	//iOptProportionalGainFor4
		aTransferPackages[15].iChannel := iParameterSet;
		aTransferPackages[15].iAddressedTarget := 8;
		aTransferPackages[15].iIndex := 249;
		
	// define end of parameter list to be uploaded by setting all variables to 0 (end criterion for FB_Upload_Multiple_Parameters)
		aTransferPackages[16].iChannel := 0;
		aTransferPackages[16].iAddressedTarget := 0;
		aTransferPackages[16].iIndex := 0;
//-----------------------------------------------------------------------------------------------------------

// Read the current status of the the motion terminal
	fbreadbitsfromword(wData:= awBusDataFromVTEM[0], iStartBit:=0, iEndBit:= 5, iValue=> iCurrentValveMode, xError=> );				// read current valve mode
//-----------------------------------------------------------------------------------------------------------

// Transition: Aborting condition when xAbort is TRUE in all States except "IDLE" , "ABORTING" and "RESETTING"
	IF xAbort = TRUE AND NOT(iState = 10 AND xExecute = FALSE) AND iState <> 80 AND iState <> 100 THEN
		xStateChange := TRUE;	// Leaving current state
		iState := 80;	// Choosing next state, here: ABORTING
	END_IF
//-----------------------------------------------------------------------------------------------------------

// local state machine
	CASE iState OF
		10:	// IDLE
			// code that is executed only in the first cycle of this state
				IF xStateChange = TRUE THEN
					xStateChange := FALSE;
					iResponse := eTransferResponse.ready_for_new_transfer;
					xDone := FALSE;
					xError := FALSE;
					xBusy := FALSE;
					xAborted := FALSE;
				END_IF
			//-----------------------------------------------------------------------------------------------------------
			
			// code that is repeated every cycle in this state
				iCommandNumber := 0;
			//-----------------------------------------------------------------------------------------------------------
			
			// Transition
			IF xExecute = TRUE THEN
				xStateChange := TRUE;
				iState := 20;
			END_IF
			//-----------------------------------------------------------------------------------------------------------
		
		20:	// RESETTING VALVE MODE TO 61
			// code that is executed only in the first cycle of this state
				IF xStateChange = TRUE THEN
					xStateChange := FALSE;
					iResponse := eTransferResponse.preparing_transfer;
					xDone := FALSE;
					xError := FALSE;
					xBusy := TRUE;
					xAborted := FALSE;
				END_IF
			//-----------------------------------------------------------------------------------------------------------
			
			// code that is repeated every cycle in this state	
				IF iCurrentValveMode = 63 THEN
					iCommandNumber := 5;	// exit transfer mode
				ELSIF iCurrentValveMode <> 61 AND iCurrentValveMode <> 63 THEN
					iCommandNumber := 6;	// stop running motion apps
				END_IF 
			//-----------------------------------------------------------------------------------------------------------
			
			// Transition
				IF iCurrentValveMode = 61 THEN
					xStateChange := TRUE;	// Leave this state
					iState := 30;
					iCommandNumber := 30;			
				END_IF
			//-----------------------------------------------------------------------------------------------------------
		
		30:	// READING PARAMETER VALUES
			// code that is executed only in the first cycle of this state
				IF xStateChange = TRUE THEN
					xStateChange := FALSE;
					iResponse := eTransferResponse.transferring;
					xDone := FALSE;
					xError := FALSE;
					xBusy := TRUE;
					xAborted := FALSE;
				END_IF
			//-----------------------------------------------------------------------------------------------------------
			
			// code that is repeated every cycle in this state
				iCommandNumber := 30;		// read parameter values
			//-----------------------------------------------------------------------------------------------------------
			
			// Transition
				IF fbuploadMultipleParameters.xExecute = TRUE AND fbuploadMultipleParameters.xUploadDone = TRUE AND fbuploadMultipleParameters.xUploadError = FALSE THEN	// Upload Done
					xStateChange := TRUE;
					iState := 40;	// Write parameter values to outputs
				ELSIF fbuploadMultipleParameters.xExecute = TRUE AND fbuploadMultipleParameters.xUploadDone = FALSE AND fbuploadMultipleParameters.xUploadError = TRUE THEN	// Error during update
					xStateChange := TRUE;
					iState := 70;	// ERROR
					iResponse := fbuploadMultipleParameters.iResponse;
				END_IF
			//-----------------------------------------------------------------------------------------------------------
		
		40:	// WRITE PARAMETER VALUES TO OUTPUTS
			// code that is executed only in the first cycle of this state
				IF xStateChange = TRUE THEN
					xStateChange := FALSE;
					iResponse := eTransferResponse.transferring;
					xDone := FALSE;
					xError := FALSE;
					xBusy := TRUE;
					xAborted := FALSE;
				END_IF
			//-----------------------------------------------------------------------------------------------------------
			
			// code that is repeated every cycle in this state
				iTubingLengthAt2			:= aTransferPackages[0].iTransferValue;
				iTubingLengthAt4			:= aTransferPackages[1].iTransferValue;
				iTubingInnerDiameterAt2		:= aTransferPackages[2].iTransferValue;
				iTubingInnerDiameterAt4		:= aTransferPackages[3].iTransferValue;
				iDriveType					:= aTransferPackages[4].iTransferValue;
				iDriveStroke				:= aTransferPackages[5].iTransferValue;
				iInstallationPositionDrive	:= aTransferPackages[6].iTransferValue;
				iLoadRetracting				:= aTransferPackages[7].iTransferValue;
				iLoadAdvancing				:= aTransferPackages[8].iTransferValue;
				iMomentOfInertiaRetracting	:= aTransferPackages[9].iTransferValue;
				iMomentOfInertiaAdvancing	:= aTransferPackages[10].iTransferValue;
				iSoftStartFunction			:= aTransferPackages[11].iTransferValue;
				iInPortRetracted_optional	:= aTransferPackages[12].iTransferValue;
				iInPortAdvanced_optional	:= aTransferPackages[13].iTransferValue;
				iOptProportionalGainFor2	:= aTransferPackages[14].iTransferValue;
				iOptProportionalGainFor4	:= aTransferPackages[15].iTransferValue;
			//-----------------------------------------------------------------------------------------------------------
			
			// Transition
				xStateChange := TRUE;
				iState := 50;
				iCommandNumber := 40;
			//-----------------------------------------------------------------------------------------------------------
		
		50:	// DONE
			// code that is executed only in the first cycle of this state
				IF xStateChange = TRUE THEN
					xStateChange := FALSE;
					iResponse := eTransferResponse.transfer_successful;
					xDone := TRUE;
					xError := FALSE;
					xBusy := FALSE;
					xAborted := FALSE;
				END_IF
			//-----------------------------------------------------------------------------------------------------------
			
			// code that is repeated every cycle in this state	
				IF fbuploadMultipleParameters.xExecute = FALSE  AND fbuploadMultipleParameters.xUploadDone = FALSE AND fbuploadMultipleParameters.xUploadError = FALSE AND iCurrentValveMode = 63 THEN		//FB_UploadMultipleParameters was reset
					iCommandNumber := 5;	// exit transfer mode
				END_IF
			//-----------------------------------------------------------------------------------------------------------
			
			// Transition
				IF fbuploadMultipleParameters.xExecute = FALSE  AND fbuploadMultipleParameters.xUploadDone = FALSE AND fbuploadMultipleParameters.xUploadError = FALSE AND xExecute = FALSE THEN
					xStateChange := TRUE;
					iState := 100;
				END_IF
			//-----------------------------------------------------------------------------------------------------------
			
		70:	// ERROR
			// code that is executed only in the first cycle of this state
				IF xStateChange = TRUE THEN
					xStateChange := FALSE;
					//iResponse := eTransferResponse.communication_failed;	// set within the transition of the last state
					xDone := FALSE;
					xError := TRUE;
					xBusy := FALSE;
					xAborted := FALSE;
				END_IF
			//-----------------------------------------------------------------------------------------------------------
			
			// code that is repeated every cycle in this state	
			//-----------------------------------------------------------------------------------------------------------
			
			// Transition
				IF xExecute = FALSE AND xAbort = FALSE THEN
					xStateChange := TRUE;
					iState := 100;
				END_IF
			//-----------------------------------------------------------------------------------------------------------
			
		80:	// ABORTING
			// code that is executed only in the first cycle of this state
				IF xStateChange = TRUE THEN
					xStateChange := FALSE;
					iResponse := eTransferResponse.aborting;
					xBusy := FALSE;
					xDone := FALSE;
					xError := FALSE;
					xAborted := TRUE;
				END_IF
			//-----------------------------------------------------------------------------------------------------------
			
			// code that is repeated every cycle in this state
				IF iCurrentValveMode = 63 THEN
					iCommandNumber := 5;	// exit transfer mode
				ELSIF iCurrentValveMode <> 61 AND iCurrentValveMode <> 63 THEN
					iCommandNumber := 6;	// stop running motion apps
				ELSE
					iCommandNumber := 0; 
				END_IF
			//-----------------------------------------------------------------------------------------------------------
			
			// Transition
				IF xAbort = FALSE AND xExecute = FALSE AND iCurrentValveMode = 61 THEN
					xStateChange := TRUE;
					iState := 100;
				END_IF
			//-----------------------------------------------------------------------------------------------------------

		100:	// RESETTING FUNCTION BLOCK AND VALVE
			// code that is executed only in the first cycle of this state
				IF xStateChange = TRUE THEN
					xStateChange := FALSE;
					iResponse := eTransferResponse.resetting;
					xDone := FALSE;
					xError := FALSE;
					xBusy := FALSE;
					xAborted := FALSE;
				END_IF
			//-----------------------------------------------------------------------------------------------------------
			
			// code that is repeated every cycle in this state	
				IF iCurrentValveMode = 63 THEN
					iCommandNumber := 5;	// exit transfer mode
				ELSIF iCurrentValveMode <> 61 AND iCurrentValveMode <> 63 THEN
					iCommandNumber := 6;	// stop running motion apps
				END_IF
				
				// reset funktion block fbreadmultipleparameters
				// not done via command number because this is used to reset valve
					fbuploadMultipleParameters(
						awBusDataFromVTEM:= awBusDataFromVTEM, 
						awBusDataToVTEM:= awBusDataToVTEM, 
						xExecute:= FALSE, 
						iResponse=> , 
						iCurrentValue=> , 
						xUploadDone=> , 
						xUploadError=> , 
						aTransferPackages:= aTransferPackages);
				
				// reset parameter outputs
					iParameterSet				:= 1;

					iTubingLengthAt2			:= 0;
					iTubingLengthAt4			:= 0;
					iTubingInnerDiameterAt2		:= 0;
					iTubingInnerDiameterAt4		:= 0;
					iDriveType					:= 0;
					iDriveStroke				:= 0;
					iInstallationPositionDrive	:= 0;
					iLoadRetracting				:= 0;
					iLoadAdvancing				:= 0;
					iMomentOfInertiaRetracting	:= 0;
					iMomentOfInertiaAdvancing	:= 0;
					iSoftStartFunction			:= 0;
					iInPortRetracted_optional	:= 0;
					iInPortAdvanced_optional	:= 0;
					iOptProportionalGainFor2	:= 0;
					iOptProportionalGainFor4	:= 0;
				
				// reset parameter array
					FOR iCounterResetArray := 0 TO 100 BY 1 DO
						aTransferPackages[iCounterResetArray].iChannel := 0;
						aTransferPackages[iCounterResetArray].iAddressedTarget := 0;
						aTransferPackages[iCounterResetArray].iIndex := 0;
						aTransferPackages[iCounterResetArray].iTransferValue := 0;
					END_FOR
					
					iCounterResetArray := 0;
					xFirstCycle := TRUE;
			//-----------------------------------------------------------------------------------------------------------
			
			// Transition
				IF iCurrentValveMode = 61 THEN
					iCommandNumber := 6; // Last command to send before the FB is in IDLE
					xStateChange := TRUE;
					iState := 10;
				END_IF
			//-----------------------------------------------------------------------------------------------------------
			
	END_CASE
//-----------------------------------------------------------------------------------------------------------

// Command section
	CASE iCommandNumber OF
		0:	// IDLE
			;
		
		5:	// EXIT TRANSFER MODE
			fbwritevaluetoword(iValue:=63, iStartBit:=0, iEndBit:=5, wDataWord:=awBusDataToVTEM[0], xError=> );							// Valve Mode = 63
			fbwritevaluetoword(iValue:=0, iStartBit:=6, iEndBit:=7, wDataWord:=awBusDataToVTEM[0], xError=> );							// 0 (unused)
			fbwritevaluetoword(iValue:=0, iStartBit:=8, iEndBit:=12, wDataWord:=awBusDataToVTEM[0], xError=> );							// Channel = 0 (ignored)
			fbwritevaluetoword(iValue:=3, iStartBit:=13, iEndBit:=15, wDataWord:=awBusDataToVTEM[0], xError=> );						// Transfer Control = 3 (Exit transfer mode)
			fbwritevaluetoword(iValue:=0, iStartBit:=0, iEndBit:=7, wDataWord:=awBusDataToVTEM[1], xError=> );							// Addressed Target = 0 (ignored)
			fbwritevaluetoword(iValue:=0, iStartBit:=8, iEndBit:=15, wDataWord:=awBusDataToVTEM[1], xError=> );							// Index = 0 (ignored)
			fbwritevaluetoword(iValue:=0, iStartBit:=0, iEndBit:=15, wDataWord:=awBusDataToVTEM[2], xError=> );							// Value = 0 (ignored)
			
		6:	// STOP RUNNING MOTION APP
			fbwritevaluetoword(iValue:=61, iStartBit:=0, iEndBit:=5, wDataWord:=awBusDataToVTEM[0], xError=> );							// Valve Mode = 61 (stop)
			fbwritevaluetoword(iValue:=0, iStartBit:=6, iEndBit:=7, wDataWord:=awBusDataToVTEM[0], xError=> );							// App Control = 0 (unused)
			fbwritevaluetoword(iValue:=0, iStartBit:=8, iEndBit:=15, wDataWord:=awBusDataToVTEM[0], xError=> );							// App Option = 0 (unused)
			fbwritevaluetoword(iValue:=0, iStartBit:=0, iEndBit:=15, wDataWord:=awBusDataToVTEM[1], xError=> );							// Setpoint Value 1 = 0 (unused)
			fbwritevaluetoword(iValue:=0, iStartBit:=0, iEndBit:=15, wDataWord:=awBusDataToVTEM[2], xError=> );							// Setpoint Value 2 = 0 (unused)
		
		30:	// RUN FB_UPLOADMULTIPLEPARAMETERS
			fbuploadMultipleParameters(
				awBusDataFromVTEM:= awBusDataFromVTEM, 
				awBusDataToVTEM:= awBusDataToVTEM, 
				xExecute:= TRUE, 
				iResponse=> , 
				iCurrentValue=> , 
				xUploadDone=> , 
				xUploadError=> , 
				aTransferPackages:= aTransferPackages);

		40:	// RESET FB_UPLOADMULTIPLEPARAMETERS
			fbuploadMultipleParameters(
				awBusDataFromVTEM:= awBusDataFromVTEM, 
				awBusDataToVTEM:= awBusDataToVTEM, 
				xExecute:= FALSE, 
				iResponse=> , 
				iCurrentValue=> , 
				xUploadDone=> , 
				xUploadError=> , 
				aTransferPackages:= aTransferPackages);
	END_CASE
//-----------------------------------------------------------------------------------------------------------

END_FUNCTION_BLOCK

// Transfermode/specific_MA_config/FB_Read_config_MA_10
/// This function block can be used to upload the configuration of Motion App 10 ("Flow control").
/// The specific parameters of this Motion App are the outputs of this FB
/// The function block uses the transfer mode to read this configuration from the Motion Terminal
/// and indicates the state of the upload process at the output iResponse.

FUNCTION_BLOCK FB_Read_config_MA_10
VAR_INPUT
	awBusDataFromVTEM 				: ARRAY [0..2] OF WORD;		// array of 3 words of process data received from the Motion Terminal
END_VAR
	
VAR_IN_OUT
	awBusDataToVTEM 				: ARRAY [0..2] OF WORD; 	// array of 3 words of process data sent to the Motion Terminal
END_VAR

VAR_INPUT
	xExecute 						: BOOL; 					// rising edge starts the reading process, falling edge resets the function block after reading is done
	xAbort							: BOOL;						// rising edge aborts the reading process
	iParameterSet					: INT := 1; 				// the parameter set to be read from, 1 by default
END_VAR                     		

VAR_OUTPUT                  		
	// system parameters
		iOperatingMedium			: eMA10OperatingMedium;		// Type and condition of the operating medium (values see eMA10OperatingMedium)
		iInPortFlowRate2_optional	: INT;						// Sensor port for flow rate at (2) (required for closed-loop controlled operating mode, value is number of the slot (beginning from 0 and including valve slots) * 10 + number of the port 
		iInPortFlowRate4_optional	: INT;						// Sensor port for flow rate at (4) (required for closed-loop controlled operating mode, value is number of the slot (beginning from 0 and including valve slots) * 10 + number of the port
		iInPortRetracted_optional	: INT;						// Sensor port for detection of end position at pressurisation of outlet port 2 (retracted), value is number of the slot (beginning from 0 and including valve slots) * 10 + number of the port
		iInPortAdvanced_optional	: INT;						// Sensor port for detection of end position at pressurisation of outlet port 4 (advanced), value is number of the slot (beginning from 0 and including valve slots) * 10 + number of the port

	// application parameters
		iCharacteristicAt2			: INT;						// Control characteristic, outlet port (2) (0 = "fast" (short tubes), 1 = medium (medium length tubes), 2 = "universal" (esp. long tubes), 3 = defined by tuning parameters (only if closed-loop control is activated for outlet port (2)))
		iCharacteristicAt4			: INT;						// Control characteristic, outlet port (4) (0 = "fast" (short tubes), 1 = medium (medium length tubes), 2 = "universal" (esp. long tubes), 3 = defined by tuning parameters (only if closed-loop control is activated for outlet port (4)))
		iOperatingMode				: INT;						// Operating mode of the Motion App (0 = (2) and (4) open-loop controlled; 1 = (2) open-loop, (4) closed-loop; 2 = (2) closed-loop, (4) open-loop; 3 = (2) and (4) closed-loop controlled) 
		xClosedLoopControl2			: BOOL;						// TRUE indicates closed-loop control for outlet port (2), FALSE is open-loop controlled operation (information is also part of parameter "iOperatingMode" and separated into an extra output for user comfort)
		xClosedLoopControl4			: BOOL;						// TRUE indicates closed-loop control for outlet port (4), FALSE is open-loop controlled operation (information is also part of parameter "iOperatingMode" and separated into an extra output for user comfort)
		
	// tuning parameters
		iOptProportionalGainFor2	: INT;						// Optional tuning parameter for the customized proportional element of the PID modulator at outlet port (2) [1 digit = 0.01 g/s/bar]
		iOptIntegralGainFor2		: INT;						// Optional tuning parameter for the customized integral element of the PID modulator at outlet port (2) [1 digit = 0.01 g/s²/bar]
		iOptRedFeedforwContrRate2	: INT;						// Optional tuning parameter for reduction of feedforward control rate of 100% for outlet port (2) [1 digit = 1%]
		iOptBoostSetpointReach2		: INT;						// Optional tuning parameter for boost to reach the setpoint value for outlet port (2) earlier, but with higher overshoot [1 digit = 1%] 
		iOptOffsetTargFRLimitInfo2	: INT;						// Optional tuning parameter for offset on the threshold value of 95% of the possible relative flow at outlet port (2) for feedback in app state, bit 5 [1 digit = 1%]
		iOptOffsetMinConsSetp2		: INT;						// Optional tuning parameter for offset to the threshold value of 25 l/min, below which a target flow rate for outlet port (2) is not considered [1 digit = 1 l/min]

		iOptProportionalGainFor4	: INT;						// Optional tuning parameter for the customized proportional element of the PID modulator at outlet port (4) [1 digit = 0.01 g/s/bar]
		iOptIntegralGainFor4		: INT;						// Optional tuning parameter for the customized integral element of the PID modulator at outlet port (4) [1 digit = 0.01 g/s²/bar]
		iOptRedFeedforwContrRate4	: INT;						// Optional tuning parameter for reduction of feedforward control rate of 100% for outlet port (4) [1 digit = 1%]
		iOptBoostSetpointReach4		: INT;						// Optional tuning parameter for boost to reach the setpoint value for outlet port (4) earlier, but with higher overshoot [1 digit = 1%] 
		iOptOffsetTargFRLimitInfo4	: INT;						// Optional tuning parameter for offset on the threshold value of 95% of the possible relative flow at outlet port (4) for feedback in app state, bit 5 [1 digit = 1%]
		iOptOffsetMinConsSetp4		: INT;						// Optional tuning parameter for offset to the threshold value of 25 l/min, below which a target flow rate for outlet port (4) is not considered [1 digit = 1 l/min]
		
	// function block response
		iResponse 					: eTransferResponse; 		// returns the status of the upload process
		xBusy						: BOOL;						// TRUE as long as the upload process is running
		xDone 						: BOOL; 					// indicates whether the upload was successfull
		xError 						: BOOL; 					// indicates whether an error occurred during the transfer
		xAborted					: BOOL;						// TRUE if the function block was canceled by xAbort	
END_VAR

VAR
	iState							: INT := 10;
	xStateChange					: BOOL;
	iCommandNumber					: INT;
	xFirstCycle						: BOOL := TRUE;				// indicator for the first cycle of the function block
	iParameterSetFC					: INT;						// value on input iParameterSet during first cycle
	
	aTransferPackages				: ARRAY [0..100] OF stTransferPackage;
	fbreadbitsfromword				: FB_Read_Bits_From_Word;
	fbuploadMultipleParameters 		: FB_Upload_Multiple_Parameters;
	fbWriteValueToWord 				: FB_Write_Value_To_Word;

	iCounterResetArray				: INT;

	iCurrentValveMode				: INT;						//
END_VAR

(*****************************************************************************************************

Festo SE & Co. KG, Esslingen
Copyright (c) 2021. All rights reserved.

Product:            Motion Terminal VTEM
Description:        Function Block to upload the parameters for Motion App 10 from the Motion Terminal

Object version:     2.00
Last change:        2021-07
======================================================================================================
                                       H I S T O R Y
======================================================================================================
Version:            2.00
Date:               2021-07
Change/Activity:    - created (#3872357)
Release:            3.5.7.237 (CODESYS 3.5.7.2, Lib version 3.7)
Author:             JEBU
======================================================================================================

*****************************************************************************************************)

// pre-check of the value for the parameter set
	IF xExecute = TRUE AND (iParameterSet < 1 OR iParameterSet > 5) THEN		// invalid input for the parameter set
		xDone := FALSE; 
		xError := TRUE; 
		iResponse := eTransferResponse.invalid_ParameterSet;
		xStateChange := TRUE;
		iState := 70;	// ERROR
	END_IF
//-----------------------------------------------------------------------------------------------------------

// check if iParameterSet was changed
	IF xExecute = TRUE AND xFirstCycle = TRUE THEN
		xFirstCycle := FALSE;
		iParameterSetFC := iParameterSet;
	END_IF
	
	IF xExecute = TRUE AND iParameterSet <> iParameterSetFC THEN
		xStateChange := TRUE;
		iState := 70;
		iResponse := eTransferResponse.FB_needs_rising_edge_xExecute;
	END_IF
//-----------------------------------------------------------------------------------------------------------

// WRITE PARAMETER INDICES INTO ARRAY
	//iOperatingMedium
		aTransferPackages[0].iChannel := iParameterSet;
		aTransferPackages[0].iAddressedTarget := 10;
		aTransferPackages[0].iIndex := 42;
	
	//iInPortFlowRate2_optional
		aTransferPackages[1].iChannel := iParameterSet;
		aTransferPackages[1].iAddressedTarget := 10;
		aTransferPackages[1].iIndex := 81;

	//iInPortFlowRate4_optional
		aTransferPackages[2].iChannel := iParameterSet;
		aTransferPackages[2].iAddressedTarget := 10;
		aTransferPackages[2].iIndex := 82;
	
	//iInPortRetracted_optional
		aTransferPackages[3].iChannel := iParameterSet;
		aTransferPackages[3].iAddressedTarget := 10;
		aTransferPackages[3].iIndex := 70;
	
	//iInPortAdvanced_optional
		aTransferPackages[4].iChannel := iParameterSet;
		aTransferPackages[4].iAddressedTarget := 10;
		aTransferPackages[4].iIndex := 71;
	
	//iCharacteristicAt2
		aTransferPackages[5].iChannel := iParameterSet;
		aTransferPackages[5].iAddressedTarget := 10;
		aTransferPackages[5].iIndex := 220;
	
	//iCharacteristicAt4
		aTransferPackages[6].iChannel := iParameterSet;
		aTransferPackages[6].iAddressedTarget := 10;
		aTransferPackages[6].iIndex := 221;
	
	//iOperatingMode
		aTransferPackages[7].iChannel := iParameterSet;
		aTransferPackages[7].iAddressedTarget := 10;
		aTransferPackages[7].iIndex := 223;
	
	//iOptProportionalGainFor2
		aTransferPackages[8].iChannel := iParameterSet;
		aTransferPackages[8].iAddressedTarget := 10;
		aTransferPackages[8].iIndex := 230;
	
	//iOptIntegralGainFor2
		aTransferPackages[9].iChannel := iParameterSet;
		aTransferPackages[9].iAddressedTarget := 10;
		aTransferPackages[9].iIndex := 231;
	
	//iOptRedFeedforwContrRate2
		aTransferPackages[10].iChannel := iParameterSet;
		aTransferPackages[10].iAddressedTarget := 10;
		aTransferPackages[10].iIndex := 232;
	
	//iOptBoostSetpointReach2
		aTransferPackages[11].iChannel := iParameterSet;
		aTransferPackages[11].iAddressedTarget := 10;
		aTransferPackages[11].iIndex := 233;
	
	//iOptOffsetTargFRLimitInfo2
		aTransferPackages[12].iChannel := iParameterSet;
		aTransferPackages[12].iAddressedTarget := 10;
		aTransferPackages[12].iIndex := 234;
	
	//iOptOffsetMinConsSetp2
		aTransferPackages[13].iChannel := iParameterSet;
		aTransferPackages[13].iAddressedTarget := 10;
		aTransferPackages[13].iIndex := 235;
	
	//iOptProportionalGainFor4
		aTransferPackages[14].iChannel := iParameterSet;
		aTransferPackages[14].iAddressedTarget := 10;
		aTransferPackages[14].iIndex := 240;
	
	//iOptIntegralGainFor4
		aTransferPackages[15].iChannel := iParameterSet;
		aTransferPackages[15].iAddressedTarget := 10;
		aTransferPackages[15].iIndex := 241;
	
	//iOptRedFeedforwContrRate4
		aTransferPackages[16].iChannel := iParameterSet;
		aTransferPackages[16].iAddressedTarget := 10;
		aTransferPackages[16].iIndex := 242;
	
	//iOptBoostSetpointReach4
		aTransferPackages[17].iChannel := iParameterSet;
		aTransferPackages[17].iAddressedTarget := 10;
		aTransferPackages[17].iIndex := 243;
	
	//iOptOffsetTargFRLimitInfo4
		aTransferPackages[18].iChannel := iParameterSet;
		aTransferPackages[18].iAddressedTarget := 10;
		aTransferPackages[18].iIndex := 244;
	
	//iOptOffsetMinConsSetp4
		aTransferPackages[19].iChannel := iParameterSet;
		aTransferPackages[19].iAddressedTarget := 10;
		aTransferPackages[19].iIndex := 245;
	
	// define end of parameter list to be uploaded by setting all variables to 0 (end criterion for FB_Upload_Multiple_Parameters)
		aTransferPackages[20].iChannel := 0;
		aTransferPackages[20].iAddressedTarget := 0;
		aTransferPackages[20].iIndex := 0;
//-----------------------------------------------------------------------------------------------------------

// Read the current status of the the motion terminal
	fbreadbitsfromword(wData:= awBusDataFromVTEM[0], iStartBit:=0, iEndBit:= 5, iValue=> iCurrentValveMode, xError=> );				// read current valve mode
//-----------------------------------------------------------------------------------------------------------

// Transition: Aborting condition when xAbort is TRUE in all States except "IDLE" , "ABORTING" and "RESETTING"
	IF xAbort = TRUE AND NOT(iState = 10 AND xExecute = FALSE) AND iState <> 80 AND iState <> 100 THEN
		xStateChange := TRUE;	// Leaving current state
		iState := 80;	// Choosing next state, here: ABORTING
	END_IF
//-----------------------------------------------------------------------------------------------------------

// local state machine
	CASE iState OF
		10:	// IDLE
			// code that is executed only in the first cycle of this state
				IF xStateChange = TRUE THEN
					xStateChange := FALSE;
					iResponse := eTransferResponse.ready_for_new_transfer;
					xDone := FALSE;
					xError := FALSE;
					xBusy := FALSE;
					xAborted := FALSE;
				END_IF
			//-----------------------------------------------------------------------------------------------------------
			
			// code that is repeated every cycle in this state
				iCommandNumber := 0;
			//-----------------------------------------------------------------------------------------------------------
			
			// Transition
			IF xExecute = TRUE THEN
				xStateChange := TRUE;
				iState := 20;
			END_IF
			//-----------------------------------------------------------------------------------------------------------
		
		20:	// RESETTING VALVE MODE TO 61
			// code that is executed only in the first cycle of this state
				IF xStateChange = TRUE THEN
					xStateChange := FALSE;
					iResponse := eTransferResponse.preparing_transfer;
					xDone := FALSE;
					xError := FALSE;
					xBusy := TRUE;
					xAborted := FALSE;
				END_IF
			//-----------------------------------------------------------------------------------------------------------
			
			// code that is repeated every cycle in this state	
				IF iCurrentValveMode = 63 THEN
					iCommandNumber := 5;	// exit transfer mode
				ELSIF iCurrentValveMode <> 61 AND iCurrentValveMode <> 63 THEN
					iCommandNumber := 6;	// stop running motion apps
				END_IF 
			//-----------------------------------------------------------------------------------------------------------
			
			// Transition
				IF iCurrentValveMode = 61 THEN
					xStateChange := TRUE;	// Leave this state
					iState := 30;
					iCommandNumber := 30;			
				END_IF
			//-----------------------------------------------------------------------------------------------------------
		
		30:	// READING PARAMETER VALUES
			// code that is executed only in the first cycle of this state
				IF xStateChange = TRUE THEN
					xStateChange := FALSE;
					iResponse := eTransferResponse.transferring;
					xDone := FALSE;
					xError := FALSE;
					xBusy := TRUE;
					xAborted := FALSE;
				END_IF
			//-----------------------------------------------------------------------------------------------------------
			
			// code that is repeated every cycle in this state
				iCommandNumber := 30;		// read parameter values
			//-----------------------------------------------------------------------------------------------------------
			
			// Transition
				IF fbuploadMultipleParameters.xExecute = TRUE AND fbuploadMultipleParameters.xUploadDone = TRUE AND fbuploadMultipleParameters.xUploadError = FALSE THEN	// Upload Done
					xStateChange := TRUE;
					iState := 40;	// Write parameter values to outputs
				ELSIF fbuploadMultipleParameters.xExecute = TRUE AND fbuploadMultipleParameters.xUploadDone = FALSE AND fbuploadMultipleParameters.xUploadError = TRUE THEN	// Error during update
					xStateChange := TRUE;
					iState := 70;	// ERROR
					iResponse := fbuploadMultipleParameters.iResponse;
				END_IF
			//-----------------------------------------------------------------------------------------------------------
		
		40:	// WRITE PARAMETER VALUES TO OUTPUTS
			// code that is executed only in the first cycle of this state
				IF xStateChange = TRUE THEN
					xStateChange := FALSE;
					iResponse := eTransferResponse.transferring;
					xDone := FALSE;
					xError := FALSE;
					xBusy := TRUE;
					xAborted := FALSE;
				END_IF
			//-----------------------------------------------------------------------------------------------------------
			
			// code that is repeated every cycle in this state
				iOperatingMedium			:= aTransferPackages[0].iTransferValue;
				iInPortFlowRate2_optional	:= aTransferPackages[1].iTransferValue;
				iInPortFlowRate4_optional	:= aTransferPackages[2].iTransferValue;
				iInPortRetracted_optional	:= aTransferPackages[3].iTransferValue;
				iInPortAdvanced_optional	:= aTransferPackages[4].iTransferValue;
				iCharacteristicAt2			:= aTransferPackages[5].iTransferValue;
				iCharacteristicAt4			:= aTransferPackages[6].iTransferValue;
				iOperatingMode				:= aTransferPackages[7].iTransferValue;
				xClosedLoopControl4			:= iOperatingMode.0;
				xClosedLoopControl2			:= iOperatingMode.1;
				iOptProportionalGainFor2	:= aTransferPackages[8].iTransferValue;
				iOptIntegralGainFor2		:= aTransferPackages[9].iTransferValue;
				iOptRedFeedforwContrRate2	:= aTransferPackages[10].iTransferValue;
				iOptBoostSetpointReach2		:= aTransferPackages[11].iTransferValue;
				iOptOffsetTargFRLimitInfo2	:= aTransferPackages[12].iTransferValue;
				iOptOffsetMinConsSetp2		:= aTransferPackages[13].iTransferValue;
				iOptProportionalGainFor4	:= aTransferPackages[14].iTransferValue;
				iOptIntegralGainFor4		:= aTransferPackages[15].iTransferValue;
				iOptRedFeedforwContrRate4	:= aTransferPackages[16].iTransferValue;
				iOptBoostSetpointReach4		:= aTransferPackages[17].iTransferValue;
				iOptOffsetTargFRLimitInfo4	:= aTransferPackages[18].iTransferValue;
				iOptOffsetMinConsSetp4		:= aTransferPackages[19].iTransferValue;
			//-----------------------------------------------------------------------------------------------------------
			
			// Transition
				xStateChange := TRUE;
				iState := 50;
				iCommandNumber := 40;
			//-----------------------------------------------------------------------------------------------------------
		
		50:	// DONE
			// code that is executed only in the first cycle of this state
				IF xStateChange = TRUE THEN
					xStateChange := FALSE;
					iResponse := eTransferResponse.transfer_successful;
					xDone := TRUE;
					xError := FALSE;
					xBusy := FALSE;
					xAborted := FALSE;
				END_IF
			//-----------------------------------------------------------------------------------------------------------
			
			// code that is repeated every cycle in this state	
				IF fbuploadMultipleParameters.xExecute = FALSE  AND fbuploadMultipleParameters.xUploadDone = FALSE AND fbuploadMultipleParameters.xUploadError = FALSE AND iCurrentValveMode = 63 THEN		//FB_UploadMultipleParameters was reset
					iCommandNumber := 5;	// exit transfer mode
				END_IF
			//-----------------------------------------------------------------------------------------------------------
			
			// Transition
				IF fbuploadMultipleParameters.xExecute = FALSE  AND fbuploadMultipleParameters.xUploadDone = FALSE AND fbuploadMultipleParameters.xUploadError = FALSE AND xExecute = FALSE THEN
					xStateChange := TRUE;
					iState := 100;
				END_IF
			//-----------------------------------------------------------------------------------------------------------
			
		70:	// ERROR
			// code that is executed only in the first cycle of this state
				IF xStateChange = TRUE THEN
					xStateChange := FALSE;
					//iResponse := eTransferResponse.communication_failed;	// set within the transition of the last state
					xDone := FALSE;
					xError := TRUE;
					xBusy := FALSE;
					xAborted := FALSE;
				END_IF
			//-----------------------------------------------------------------------------------------------------------
			
			// code that is repeated every cycle in this state	
			//-----------------------------------------------------------------------------------------------------------
			
			// Transition
				IF xExecute = FALSE AND xAbort = FALSE THEN
					xStateChange := TRUE;
					iState := 100;
				END_IF
			//-----------------------------------------------------------------------------------------------------------
			
		80:	// ABORTING
			// code that is executed only in the first cycle of this state
				IF xStateChange = TRUE THEN
					xStateChange := FALSE;
					iResponse := eTransferResponse.aborting;
					xBusy := FALSE;
					xDone := FALSE;
					xError := FALSE;
					xAborted := TRUE;
				END_IF
			//-----------------------------------------------------------------------------------------------------------
			
			// code that is repeated every cycle in this state
				IF iCurrentValveMode = 63 THEN
					iCommandNumber := 5;	// exit transfer mode
				ELSIF iCurrentValveMode <> 61 AND iCurrentValveMode <> 63 THEN
					iCommandNumber := 6;	// stop running motion apps
				ELSE
					iCommandNumber := 0; 
				END_IF
			//-----------------------------------------------------------------------------------------------------------
			
			// Transition
				IF xAbort = FALSE AND xExecute = FALSE AND iCurrentValveMode = 61 THEN
					xStateChange := TRUE;
					iState := 100;
				END_IF
			//-----------------------------------------------------------------------------------------------------------

		100:	// RESETTING FUNCTION BLOCK AND VALVE
			// code that is executed only in the first cycle of this state
				IF xStateChange = TRUE THEN
					xStateChange := FALSE;
					iResponse := eTransferResponse.resetting;
					xDone := FALSE;
					xError := FALSE;
					xBusy := FALSE;
					xAborted := FALSE;
				END_IF
			//-----------------------------------------------------------------------------------------------------------
			
			// code that is repeated every cycle in this state	
				IF iCurrentValveMode = 63 THEN
					iCommandNumber := 5;	// exit transfer mode
				ELSIF iCurrentValveMode <> 61 AND iCurrentValveMode <> 63 THEN
					iCommandNumber := 6;	// stop running motion apps
				END_IF
				
				// reset funktion block fbreadmultipleparameters
				// not done via command number because this is used to reset valve
					fbuploadMultipleParameters(
						awBusDataFromVTEM:= awBusDataFromVTEM, 
						awBusDataToVTEM:= awBusDataToVTEM, 
						xExecute:= FALSE, 
						iResponse=> , 
						iCurrentValue=> , 
						xUploadDone=> , 
						xUploadError=> , 
						aTransferPackages:= aTransferPackages);
				
				// reset parameter outputs
					iParameterSet				:= 1;

					iOperatingMedium			:= 0;
					iInPortFlowRate2_optional	:= 0;
					iInPortFlowRate4_optional	:= 0;
					iInPortRetracted_optional	:= 0;
					iInPortAdvanced_optional	:= 0;
					iCharacteristicAt2			:= 0;
					iCharacteristicAt4			:= 0;
					iOperatingMode				:= 0;
					xClosedLoopControl4			:= 0;
					xClosedLoopControl2			:= 0;
					iOptProportionalGainFor2	:= 0;
					iOptIntegralGainFor2		:= 0;
					iOptRedFeedforwContrRate2	:= 0;
					iOptBoostSetpointReach2		:= 0;
					iOptOffsetTargFRLimitInfo2	:= 0;
					iOptOffsetMinConsSetp2		:= 0;
					iOptProportionalGainFor4	:= 0;
					iOptIntegralGainFor4		:= 0;
					iOptRedFeedforwContrRate4	:= 0;
					iOptBoostSetpointReach4		:= 0;
					iOptOffsetTargFRLimitInfo4	:= 0;
					iOptOffsetMinConsSetp4		:= 0;
				
				// reset parameter array
					FOR iCounterResetArray := 0 TO 100 BY 1 DO
						aTransferPackages[iCounterResetArray].iChannel := 0;
						aTransferPackages[iCounterResetArray].iAddressedTarget := 0;
						aTransferPackages[iCounterResetArray].iIndex := 0;
						aTransferPackages[iCounterResetArray].iTransferValue := 0;
					END_FOR
					
					iCounterResetArray := 0;
					xFirstCycle := TRUE;
			//-----------------------------------------------------------------------------------------------------------
			
			// Transition
				IF iCurrentValveMode = 61 THEN
					iCommandNumber := 6; // Last command to send before the FB is in IDLE
					xStateChange := TRUE;
					iState := 10;
				END_IF
			//-----------------------------------------------------------------------------------------------------------
			
	END_CASE
//-----------------------------------------------------------------------------------------------------------

// Command section
	CASE iCommandNumber OF
		0:	// IDLE
			;
		
		5:	// EXIT TRANSFER MODE
			fbwritevaluetoword(iValue:=63, iStartBit:=0, iEndBit:=5, wDataWord:=awBusDataToVTEM[0], xError=> );							// Valve Mode = 63
			fbwritevaluetoword(iValue:=0, iStartBit:=6, iEndBit:=7, wDataWord:=awBusDataToVTEM[0], xError=> );							// 0 (unused)
			fbwritevaluetoword(iValue:=0, iStartBit:=8, iEndBit:=12, wDataWord:=awBusDataToVTEM[0], xError=> );							// Channel = 0 (ignored)
			fbwritevaluetoword(iValue:=3, iStartBit:=13, iEndBit:=15, wDataWord:=awBusDataToVTEM[0], xError=> );						// Transfer Control = 3 (Exit transfer mode)
			fbwritevaluetoword(iValue:=0, iStartBit:=0, iEndBit:=7, wDataWord:=awBusDataToVTEM[1], xError=> );							// Addressed Target = 0 (ignored)
			fbwritevaluetoword(iValue:=0, iStartBit:=8, iEndBit:=15, wDataWord:=awBusDataToVTEM[1], xError=> );							// Index = 0 (ignored)
			fbwritevaluetoword(iValue:=0, iStartBit:=0, iEndBit:=15, wDataWord:=awBusDataToVTEM[2], xError=> );							// Value = 0 (ignored)
			
		6:	// STOP RUNNING MOTION APP
			fbwritevaluetoword(iValue:=61, iStartBit:=0, iEndBit:=5, wDataWord:=awBusDataToVTEM[0], xError=> );							// Valve Mode = 61 (stop)
			fbwritevaluetoword(iValue:=0, iStartBit:=6, iEndBit:=7, wDataWord:=awBusDataToVTEM[0], xError=> );							// App Control = 0 (unused)
			fbwritevaluetoword(iValue:=0, iStartBit:=8, iEndBit:=15, wDataWord:=awBusDataToVTEM[0], xError=> );							// App Option = 0 (unused)
			fbwritevaluetoword(iValue:=0, iStartBit:=0, iEndBit:=15, wDataWord:=awBusDataToVTEM[1], xError=> );							// Setpoint Value 1 = 0 (unused)
			fbwritevaluetoword(iValue:=0, iStartBit:=0, iEndBit:=15, wDataWord:=awBusDataToVTEM[2], xError=> );							// Setpoint Value 2 = 0 (unused)
		
		30:	// RUN FB_UPLOADMULTIPLEPARAMETERS
			fbuploadMultipleParameters(
				awBusDataFromVTEM:= awBusDataFromVTEM, 
				awBusDataToVTEM:= awBusDataToVTEM, 
				xExecute:= TRUE, 
				iResponse=> , 
				iCurrentValue=> , 
				xUploadDone=> , 
				xUploadError=> , 
				aTransferPackages:= aTransferPackages);

		40:	// RESET FB_UPLOADMULTIPLEPARAMETERS
			fbuploadMultipleParameters(
				awBusDataFromVTEM:= awBusDataFromVTEM, 
				awBusDataToVTEM:= awBusDataToVTEM, 
				xExecute:= FALSE, 
				iResponse=> , 
				iCurrentValue=> , 
				xUploadDone=> , 
				xUploadError=> , 
				aTransferPackages:= aTransferPackages);
	END_CASE
//-----------------------------------------------------------------------------------------------------------

END_FUNCTION_BLOCK

// Transfermode/specific_MA_config/FB_Read_config_MA_11
/// This function block can be used to upload the configuration of Motion App 11 ("Soft stop").
/// The specific parameters of this Motion App are the outputs of this FB
/// The function block uses the transfer mode to read this configuration from the Motion Terminal
/// and indicates the state of the upload process at the output iResponse.

FUNCTION_BLOCK FB_Read_config_MA_11
VAR_INPUT
	awBusDataFromVTEM 				: ARRAY [0..2] OF WORD;		// array of 3 words of process data received from the Motion Terminal
END_VAR
	
VAR_IN_OUT
	awBusDataToVTEM 				: ARRAY [0..2] OF WORD; 	// array of 3 words of process data sent to the Motion Terminal
END_VAR

VAR_INPUT
	xExecute 						: BOOL; 					// rising edge starts the reading process, falling edge resets the function block after reading is done
	xAbort							: BOOL;						// rising edge aborts the reading process
	iParameterSet					: INT := 1; 				// the parameter set to be read from, 1 by default
END_VAR                     		

VAR_OUTPUT                  		
	// system parameters
		iDriveType 					: INT;						// type of the drive/cylinder/... that is to be operated by the valve ->  see list of drive types at support portal (www.festo.com/sp/)
	 	iDriveStroke 				: INT; 						// stroke of the drive/cylinder/... that is to be operated by the valve [1 digit = 1 mm for linear drives, 1 digit = 1° for rotary drives]
		iInstallationPositionDrive 	: INT;  	 				// inclination of the cylinder with reference to a horizontal installation position [1 digit = 0.01°, positive values = advancing upwards]
		iInPortRetracted			: INT;						// Sensor port for detection of end position at pressurisation of outlet port 2 (retracted), value is number of the slot (beginning from 0 and including valve slots) * 10 + number of the port
		iInPortAdvanced				: INT;						// Sensor port for detection of end position at pressurisation of outlet port 4 (advanced), value is number of the slot (beginning from 0 and including valve slots) * 10 + number of the port
	
	// application parameters                               	
	 	iLoadAdvancing 				: INT; 						// mass that is to be moved by the drive when advancing ((4) pressurised) [1 digit = 0.01 kg]
		iLoadRetracting 			: INT;						// mass that is to be moved by the drive when retracting ((2) pressurised) [1 digit = 0.01 kg]
		
	// function block response
		iResponse 					: eTransferResponse; 		// returns the status of the upload process
		xBusy						: BOOL;						// TRUE as long as the upload process is running
		xDone 						: BOOL; 					// indicates whether the upload was successfull
		xError 						: BOOL; 					// indicates whether an error occurred during the transfer
		xAborted					: BOOL;						// TRUE if the function block was canceled by xAbort	
END_VAR

VAR
	iState							: INT := 10;
	xStateChange					: BOOL;
	iCommandNumber					: INT;
	xFirstCycle						: BOOL := TRUE;				// indicator for the first cycle of the function block
	iParameterSetFC					: INT;						// value on input iParameterSet during first cycle
	
	aTransferPackages				: ARRAY [0..100] OF stTransferPackage;
	fbreadbitsfromword				: FB_Read_Bits_From_Word;
	fbuploadMultipleParameters 		: FB_Upload_Multiple_Parameters;
	fbWriteValueToWord 				: FB_Write_Value_To_Word;

	iCounterResetArray				: INT;

	iCurrentValveMode				: INT;						//
END_VAR

(*****************************************************************************************************

Festo SE & Co. KG, Esslingen
Copyright (c) 2021. All rights reserved.

Product:            Motion Terminal VTEM
Description:        Function Block to upload the parameters for Motion App 11 from the Motion Terminal

Object version:     2.00
Last change:        2021-07
======================================================================================================
                                       H I S T O R Y
======================================================================================================
Version:            2.00
Date:               2021-07
Change/Activity:    - created (#3872357)
Release:            3.5.7.237 (CODESYS 3.5.7.2, Lib version 3.7)
Author:             JEBU
======================================================================================================

*****************************************************************************************************)

// pre-check of the value for the parameter set
	IF xExecute = TRUE AND (iParameterSet < 1 OR iParameterSet > 5) THEN		// invalid input for the parameter set
		xDone := FALSE; 
		xError := TRUE; 
		iResponse := eTransferResponse.invalid_ParameterSet;
		xStateChange := TRUE;
		iState := 70;	// ERROR
	END_IF
//-----------------------------------------------------------------------------------------------------------

// check if iParameterSet was changed
	IF xExecute = TRUE AND xFirstCycle = TRUE THEN
		xFirstCycle := FALSE;
		iParameterSetFC := iParameterSet;
	END_IF
	
	IF xExecute = TRUE AND iParameterSet <> iParameterSetFC THEN
		xStateChange := TRUE;
		iState := 70;
		iResponse := eTransferResponse.FB_needs_rising_edge_xExecute;
	END_IF
//-----------------------------------------------------------------------------------------------------------

// WRITE PARAMETER INDICES INTO ARRAY
	//iDriveType
		aTransferPackages[0].iChannel := iParameterSet;
		aTransferPackages[0].iAddressedTarget := 11;
		aTransferPackages[0].iIndex := 20;
		
	//iDriveStroke
		aTransferPackages[1].iChannel := iParameterSet;
		aTransferPackages[1].iAddressedTarget := 11;
		aTransferPackages[1].iIndex := 21;
		
	//iInstallationPositionDrive
		aTransferPackages[2].iChannel := iParameterSet;
		aTransferPackages[2].iAddressedTarget := 11;
		aTransferPackages[2].iIndex := 60;
		
	//iLoadAdvancing
		aTransferPackages[3].iChannel := iParameterSet;
		aTransferPackages[3].iAddressedTarget := 11;
		aTransferPackages[3].iIndex := 101;
		
	//iLoadRetracting
		aTransferPackages[4].iChannel := iParameterSet;
		aTransferPackages[4].iAddressedTarget := 11;
		aTransferPackages[4].iIndex := 100;
		
	//iInPortRetract
		aTransferPackages[5].iChannel := iParameterSet;
		aTransferPackages[5].iAddressedTarget := 11;
		aTransferPackages[5].iIndex := 75;
	
	//iInPortRetract
		aTransferPackages[6].iChannel := iParameterSet;
		aTransferPackages[6].iAddressedTarget := 11;
		aTransferPackages[6].iIndex := 76;
	
	// define end of parameter list to be uploaded by setting all variables to 0 (end criterion for FB_Upload_Multiple_Parameters)
		aTransferPackages[7].iChannel := 0;
		aTransferPackages[7].iAddressedTarget := 0;
		aTransferPackages[7].iIndex := 0;
//-----------------------------------------------------------------------------------------------------------

// Read the current status of the the motion terminal
	fbreadbitsfromword(wData:= awBusDataFromVTEM[0], iStartBit:=0, iEndBit:= 5, iValue=> iCurrentValveMode, xError=> );				// read current valve mode
//-----------------------------------------------------------------------------------------------------------

// Transition: Aborting condition when xAbort is TRUE in all States except "IDLE" , "ABORTING" and "RESETTING"
	IF xAbort = TRUE AND NOT(iState = 10 AND xExecute = FALSE) AND iState <> 80 AND iState <> 100 THEN
		xStateChange := TRUE;	// Leaving current state
		iState := 80;	// Choosing next state, here: ABORTING
	END_IF
//-----------------------------------------------------------------------------------------------------------

// local state machine
	CASE iState OF
		10:	// IDLE
			// code that is executed only in the first cycle of this state
				IF xStateChange = TRUE THEN
					xStateChange := FALSE;
					iResponse := eTransferResponse.ready_for_new_transfer;
					xDone := FALSE;
					xError := FALSE;
					xBusy := FALSE;
					xAborted := FALSE;
				END_IF
			//-----------------------------------------------------------------------------------------------------------
			
			// code that is repeated every cycle in this state
				iCommandNumber := 0;
			//-----------------------------------------------------------------------------------------------------------
			
			// Transition
			IF xExecute = TRUE THEN
				xStateChange := TRUE;
				iState := 20;
			END_IF
			//-----------------------------------------------------------------------------------------------------------
		
		20:	// RESETTING VALVE MODE TO 61
			// code that is executed only in the first cycle of this state
				IF xStateChange = TRUE THEN
					xStateChange := FALSE;
					iResponse := eTransferResponse.preparing_transfer;
					xDone := FALSE;
					xError := FALSE;
					xBusy := TRUE;
					xAborted := FALSE;
				END_IF
			//-----------------------------------------------------------------------------------------------------------
			
			// code that is repeated every cycle in this state	
				IF iCurrentValveMode = 63 THEN
					iCommandNumber := 5;	// exit transfer mode
				ELSIF iCurrentValveMode <> 61 AND iCurrentValveMode <> 63 THEN
					iCommandNumber := 6;	// stop running motion apps
				END_IF 
			//-----------------------------------------------------------------------------------------------------------
			
			// Transition
				IF iCurrentValveMode = 61 THEN
					xStateChange := TRUE;	// Leave this state
					iState := 30;
					iCommandNumber := 30;			
				END_IF
			//-----------------------------------------------------------------------------------------------------------
		
		30:	// READING PARAMETER VALUES
			// code that is executed only in the first cycle of this state
				IF xStateChange = TRUE THEN
					xStateChange := FALSE;
					iResponse := eTransferResponse.transferring;
					xDone := FALSE;
					xError := FALSE;
					xBusy := TRUE;
					xAborted := FALSE;
				END_IF
			//-----------------------------------------------------------------------------------------------------------
			
			// code that is repeated every cycle in this state
				iCommandNumber := 30;		// read parameter values
			//-----------------------------------------------------------------------------------------------------------
			
			// Transition
				IF fbuploadMultipleParameters.xExecute = TRUE AND fbuploadMultipleParameters.xUploadDone = TRUE AND fbuploadMultipleParameters.xUploadError = FALSE THEN	// Upload Done
					xStateChange := TRUE;
					iState := 40;	// Write parameter values to outputs
				ELSIF fbuploadMultipleParameters.xExecute = TRUE AND fbuploadMultipleParameters.xUploadDone = FALSE AND fbuploadMultipleParameters.xUploadError = TRUE THEN	// Error during update
					xStateChange := TRUE;
					iState := 70;	// ERROR
					iResponse := fbuploadMultipleParameters.iResponse;
				END_IF
			//-----------------------------------------------------------------------------------------------------------
		
		40:	// WRITE PARAMETER VALUES TO OUTPUTS
			// code that is executed only in the first cycle of this state
				IF xStateChange = TRUE THEN
					xStateChange := FALSE;
					iResponse := eTransferResponse.transferring;
					xDone := FALSE;
					xError := FALSE;
					xBusy := TRUE;
					xAborted := FALSE;
				END_IF
			//-----------------------------------------------------------------------------------------------------------
			
			// code that is repeated every cycle in this state
				iDriveType					:= aTransferPackages[0].iTransferValue;
				iDriveStroke				:= aTransferPackages[1].iTransferValue;
				iInstallationPositionDrive	:= aTransferPackages[2].iTransferValue;
				iLoadAdvancing				:= aTransferPackages[3].iTransferValue;
				iLoadRetracting				:= aTransferPackages[4].iTransferValue;
				iInPortRetracted			:= aTransferPackages[5].iTransferValue;
				iInPortAdvanced				:= aTransferPackages[6].iTransferValue;
			//-----------------------------------------------------------------------------------------------------------
			
			// Transition
				xStateChange := TRUE;
				iState := 50;
				iCommandNumber := 40;
			//-----------------------------------------------------------------------------------------------------------
		
		50:	// DONE
			// code that is executed only in the first cycle of this state
				IF xStateChange = TRUE THEN
					xStateChange := FALSE;
					iResponse := eTransferResponse.transfer_successful;
					xDone := TRUE;
					xError := FALSE;
					xBusy := FALSE;
					xAborted := FALSE;
				END_IF
			//-----------------------------------------------------------------------------------------------------------
			
			// code that is repeated every cycle in this state	
				IF fbuploadMultipleParameters.xExecute = FALSE  AND fbuploadMultipleParameters.xUploadDone = FALSE AND fbuploadMultipleParameters.xUploadError = FALSE AND iCurrentValveMode = 63 THEN		//FB_UploadMultipleParameters was reset
					iCommandNumber := 5;	// exit transfer mode
				END_IF
			//-----------------------------------------------------------------------------------------------------------
			
			// Transition
				IF fbuploadMultipleParameters.xExecute = FALSE  AND fbuploadMultipleParameters.xUploadDone = FALSE AND fbuploadMultipleParameters.xUploadError = FALSE AND xExecute = FALSE THEN
					xStateChange := TRUE;
					iState := 100;
				END_IF
			//-----------------------------------------------------------------------------------------------------------
			
		70:	// ERROR
			// code that is executed only in the first cycle of this state
				IF xStateChange = TRUE THEN
					xStateChange := FALSE;
					//iResponse := eTransferResponse.communication_failed;	// set within the transition of the last state
					xDone := FALSE;
					xError := TRUE;
					xBusy := FALSE;
					xAborted := FALSE;
				END_IF
			//-----------------------------------------------------------------------------------------------------------
			
			// code that is repeated every cycle in this state	
			//-----------------------------------------------------------------------------------------------------------
			
			// Transition
				IF xExecute = FALSE AND xAbort = FALSE THEN
					xStateChange := TRUE;
					iState := 100;
				END_IF
			//-----------------------------------------------------------------------------------------------------------
			
		80:	// ABORTING
			// code that is executed only in the first cycle of this state
				IF xStateChange = TRUE THEN
					xStateChange := FALSE;
					iResponse := eTransferResponse.aborting;
					xBusy := FALSE;
					xDone := FALSE;
					xError := FALSE;
					xAborted := TRUE;
				END_IF
			//-----------------------------------------------------------------------------------------------------------
			
			// code that is repeated every cycle in this state
				IF iCurrentValveMode = 63 THEN
					iCommandNumber := 5;	// exit transfer mode
				ELSIF iCurrentValveMode <> 61 AND iCurrentValveMode <> 63 THEN
					iCommandNumber := 6;	// stop running motion apps
				ELSE
					iCommandNumber := 0; 
				END_IF
			//-----------------------------------------------------------------------------------------------------------
			
			// Transition
				IF xAbort = FALSE AND xExecute = FALSE AND iCurrentValveMode = 61 THEN
					xStateChange := TRUE;
					iState := 100;
				END_IF
			//-----------------------------------------------------------------------------------------------------------

		100:	// RESETTING FUNCTION BLOCK AND VALVE
			// code that is executed only in the first cycle of this state
				IF xStateChange = TRUE THEN
					xStateChange := FALSE;
					iResponse := eTransferResponse.resetting;
					xDone := FALSE;
					xError := FALSE;
					xBusy := FALSE;
					xAborted := FALSE;
				END_IF
			//-----------------------------------------------------------------------------------------------------------
			
			// code that is repeated every cycle in this state	
				IF iCurrentValveMode = 63 THEN
					iCommandNumber := 5;	// exit transfer mode
				ELSIF iCurrentValveMode <> 61 AND iCurrentValveMode <> 63 THEN
					iCommandNumber := 6;	// stop running motion apps
				END_IF
				
				// reset funktion block fbreadmultipleparameters
				// not done via command number because this is used to reset valve
					fbuploadMultipleParameters(
						awBusDataFromVTEM:= awBusDataFromVTEM, 
						awBusDataToVTEM:= awBusDataToVTEM, 
						xExecute:= FALSE, 
						iResponse=> , 
						iCurrentValue=> , 
						xUploadDone=> , 
						xUploadError=> , 
						aTransferPackages:= aTransferPackages);
				
				// reset parameter outputs
					iParameterSet				:= 1;

					iDriveType					:= 0;
					iDriveStroke				:= 0;
					iInstallationPositionDrive	:= 0;
					iLoadAdvancing				:= 0;
					iLoadRetracting				:= 0;
					iInPortRetracted			:= 0;
					iInPortAdvanced				:= 0;
				
				// reset parameter array
					FOR iCounterResetArray := 0 TO 100 BY 1 DO
						aTransferPackages[iCounterResetArray].iChannel := 0;
						aTransferPackages[iCounterResetArray].iAddressedTarget := 0;
						aTransferPackages[iCounterResetArray].iIndex := 0;
						aTransferPackages[iCounterResetArray].iTransferValue := 0;
					END_FOR
					
					iCounterResetArray := 0;
					xFirstCycle := TRUE;
			//-----------------------------------------------------------------------------------------------------------
			
			// Transition
				IF iCurrentValveMode = 61 THEN
					iCommandNumber := 6; // Last command to send before the FB is in IDLE
					xStateChange := TRUE;
					iState := 10;
				END_IF
			//-----------------------------------------------------------------------------------------------------------
			
	END_CASE
//-----------------------------------------------------------------------------------------------------------

// Command section
	CASE iCommandNumber OF
		0:	// IDLE
			;
		
		5:	// EXIT TRANSFER MODE
			fbwritevaluetoword(iValue:=63, iStartBit:=0, iEndBit:=5, wDataWord:=awBusDataToVTEM[0], xError=> );							// Valve Mode = 63
			fbwritevaluetoword(iValue:=0, iStartBit:=6, iEndBit:=7, wDataWord:=awBusDataToVTEM[0], xError=> );							// 0 (unused)
			fbwritevaluetoword(iValue:=0, iStartBit:=8, iEndBit:=12, wDataWord:=awBusDataToVTEM[0], xError=> );							// Channel = 0 (ignored)
			fbwritevaluetoword(iValue:=3, iStartBit:=13, iEndBit:=15, wDataWord:=awBusDataToVTEM[0], xError=> );						// Transfer Control = 3 (Exit transfer mode)
			fbwritevaluetoword(iValue:=0, iStartBit:=0, iEndBit:=7, wDataWord:=awBusDataToVTEM[1], xError=> );							// Addressed Target = 0 (ignored)
			fbwritevaluetoword(iValue:=0, iStartBit:=8, iEndBit:=15, wDataWord:=awBusDataToVTEM[1], xError=> );							// Index = 0 (ignored)
			fbwritevaluetoword(iValue:=0, iStartBit:=0, iEndBit:=15, wDataWord:=awBusDataToVTEM[2], xError=> );							// Value = 0 (ignored)
			
		6:	// STOP RUNNING MOTION APP
			fbwritevaluetoword(iValue:=61, iStartBit:=0, iEndBit:=5, wDataWord:=awBusDataToVTEM[0], xError=> );							// Valve Mode = 61 (stop)
			fbwritevaluetoword(iValue:=0, iStartBit:=6, iEndBit:=7, wDataWord:=awBusDataToVTEM[0], xError=> );							// App Control = 0 (unused)
			fbwritevaluetoword(iValue:=0, iStartBit:=8, iEndBit:=15, wDataWord:=awBusDataToVTEM[0], xError=> );							// App Option = 0 (unused)
			fbwritevaluetoword(iValue:=0, iStartBit:=0, iEndBit:=15, wDataWord:=awBusDataToVTEM[1], xError=> );							// Setpoint Value 1 = 0 (unused)
			fbwritevaluetoword(iValue:=0, iStartBit:=0, iEndBit:=15, wDataWord:=awBusDataToVTEM[2], xError=> );							// Setpoint Value 2 = 0 (unused)
		
		30:	// RUN FB_UPLOADMULTIPLEPARAMETERS
			fbuploadMultipleParameters(
				awBusDataFromVTEM:= awBusDataFromVTEM, 
				awBusDataToVTEM:= awBusDataToVTEM, 
				xExecute:= TRUE, 
				iResponse=> , 
				iCurrentValue=> , 
				xUploadDone=> , 
				xUploadError=> , 
				aTransferPackages:= aTransferPackages);

		40:	// RESET FB_UPLOADMULTIPLEPARAMETERS
			fbuploadMultipleParameters(
				awBusDataFromVTEM:= awBusDataFromVTEM, 
				awBusDataToVTEM:= awBusDataToVTEM, 
				xExecute:= FALSE, 
				iResponse=> , 
				iCurrentValue=> , 
				xUploadDone=> , 
				xUploadError=> , 
				aTransferPackages:= aTransferPackages);
	END_CASE
//-----------------------------------------------------------------------------------------------------------

END_FUNCTION_BLOCK

// Transfermode/specific_MA_config/FB_Read_config_MA_12
/// This function block can be used to upload the configuration of Motion App 12 ("Leakage diagnostics").
/// The specific parameters of this Motion App are the outputs of this FB
/// The function block uses the transfer mode to read this configuration from the Motion Terminal
/// and indicates the state of the upload process at the output iResponse.

FUNCTION_BLOCK FB_Read_config_MA_12
VAR_INPUT
	awBusDataFromVTEM 				: ARRAY [0..2] OF WORD;		// array of 3 words of process data received from the Motion Terminal
END_VAR
	
VAR_IN_OUT
	awBusDataToVTEM 				: ARRAY [0..2] OF WORD; 	// array of 3 words of process data sent to the Motion Terminal
END_VAR

VAR_INPUT
	xExecute 						: BOOL; 					// rising edge starts the reading process, falling edge resets the function block after reading is done
	xAbort							: BOOL;						// rising edge aborts the reading process
	iParameterSet					: INT := 1; 				// the parameter set to be read from, 1 by default
END_VAR                     		

VAR_OUTPUT                  		
	// system parameters
		iTubingLengthAt2 			: INT; 						// length of the tubing connected to outlet port 2 of the valve [1 digit = 1 mm]
	 	iTubingLengthAt4 			: INT;						// length of the tubing connected to outlet port 4 of the valve [1 digit = 1 mm]
	 	iTubingInnerDiameterAt2		: INT;  					// inner diameter of the tubing connected to outlet port 2 of the valve [1 digit = 0.01mm]
	 	iTubingInnerDiameterAt4		: INT;						// inner diameter of the tubing connected to outlet port 4 of the valve [1 digit = 0.01mm]
	 	iDriveType 					: INT;						// type of the drive/cylinder/... that is to be operated by the valve ->  see list of drive types at support portal (www.festo.com/sp/)
	 	iDriveStroke 				: INT; 						// stroke of the drive/cylinder/... that is to be operated by the valve [1 digit = 1 mm for linear drives, 1 digit = 1° for rotary drives]
		iVolumeAt2 					: INT; 						// size/capacity of the volume connected to outlet port 2 of the valve [1 digit = 0.001 l]
		iVolumeAt4 					: INT;						// size/capacity of the volume connected to outlet port 4 of the valve [1 digit = 0.001 l]
		iInstallationPositionDrive 	: INT;  	 				// inclination of the cylinder with reference to a horizontal installation position [1 digit = 0.01°, positive values = advancing upwards]

	// application parameters                               	
		iLoadRetracting 			: INT;						// mass that is to be moved by the drive when retracting ((2) pressurised) [1 digit = 0.01 kg]
	 	iLoadAdvancing 				: INT; 						// mass that is to be moved by the drive when advancing ((4) pressurised) [1 digit = 0.01 kg]
		iMomentOfInertiaRetracting	: INT;						// Moment of inertia during for swivel drives when retratcting ((2) pressirised) [1 digit = 1 kg cm³]
		iMomentOfInertiaAdvancing	: INT;						// Moment of inertia during for swivel drives when advancing ((4) pressirised) [1 digit = 1 kg cm³]
		iMaxLeakageForStatusGood 	: INT;						// allowed deviation regarding reference value for status "Good" [1 digit = 0.1 l/h]
		iMaxLeakageForStatusWarning : INT;						// allowed deviation regarding reference value for status "Warning" [1 digit = 0.1 l/h]
	 	iMaxLeakageForStatusCritical: INT; 						// allowed deviation regarding reference value for status "Critical" [1 digit = 0.1 l/h]
		
	// function block response
		iResponse 					: eTransferResponse; 		// returns the status of the upload process
		xBusy						: BOOL;						// TRUE as long as the upload process is running
		xDone 						: BOOL; 					// indicates whether the upload was successfull
		xError 						: BOOL; 					// indicates whether an error occurred during the transfer
		xAborted					: BOOL;						// TRUE if the function block was canceled by xAbort	
END_VAR

VAR
	iState							: INT := 10;
	xStateChange					: BOOL;
	iCommandNumber					: INT;
	xFirstCycle						: BOOL := TRUE;				// indicator for the first cycle of the function block
	iParameterSetFC					: INT;						// value on input iParameterSet during first cycle
	
	aTransferPackages				: ARRAY [0..100] OF stTransferPackage;
	fbreadbitsfromword				: FB_Read_Bits_From_Word;
	fbuploadMultipleParameters 		: FB_Upload_Multiple_Parameters;
	fbWriteValueToWord 				: FB_Write_Value_To_Word;

	iCounterResetArray				: INT;

	iCurrentValveMode				: INT;						//
END_VAR

(*****************************************************************************************************

Festo SE & Co. KG, Esslingen
Copyright (c) 2021. All rights reserved.

Product:            Motion Terminal VTEM
Description:        Function Block to upload the parameters for Motion App 12 from the Motion Terminal

Object version:     2.00
Last change:        2021-07
======================================================================================================
                                       H I S T O R Y
======================================================================================================
Version:            2.00
Date:               2021-07
Change/Activity:    - created (#3872357)
Release:            3.5.7.237 (CODESYS 3.5.7.2, Lib version 3.7)
Author:             JEBU
======================================================================================================

*****************************************************************************************************)

// pre-check of the value for the parameter set
	IF xExecute = TRUE AND (iParameterSet < 1 OR iParameterSet > 5) THEN		// invalid input for the parameter set
		xDone := FALSE; 
		xError := TRUE; 
		iResponse := eTransferResponse.invalid_ParameterSet;
		xStateChange := TRUE;
		iState := 70;	// ERROR
	END_IF
//-----------------------------------------------------------------------------------------------------------

// check if iParameterSet was changed
	IF xExecute = TRUE AND xFirstCycle = TRUE THEN
		xFirstCycle := FALSE;
		iParameterSetFC := iParameterSet;
	END_IF
	
	IF xExecute = TRUE AND iParameterSet <> iParameterSetFC THEN
		xStateChange := TRUE;
		iState := 70;
		iResponse := eTransferResponse.FB_needs_rising_edge_xExecute;
	END_IF
//-----------------------------------------------------------------------------------------------------------

// WRITE PARAMETER INDICES INTO ARRAY
	//iTubingLengthAt2
		aTransferPackages[0].iChannel := iParameterSet;
		aTransferPackages[0].iAddressedTarget := 12;
		aTransferPackages[0].iIndex := 12;
		
	//iTubingLengthAt4
		aTransferPackages[1].iChannel := iParameterSet;
		aTransferPackages[1].iAddressedTarget := 12;
		aTransferPackages[1].iIndex := 13;
		
	//iTubingInnerDiameterAt2
		aTransferPackages[2].iChannel := iParameterSet;
		aTransferPackages[2].iAddressedTarget := 12;
		aTransferPackages[2].iIndex := 14;
		
	//iTubingInnerDiameterAt4
		aTransferPackages[3].iChannel := iParameterSet;
		aTransferPackages[3].iAddressedTarget := 12;
		aTransferPackages[3].iIndex := 15;
		
	//iDriveType
		aTransferPackages[4].iChannel := iParameterSet;
		aTransferPackages[4].iAddressedTarget := 12;
		aTransferPackages[4].iIndex := 20;
		
	//iDriveStroke
		aTransferPackages[5].iChannel := iParameterSet;
		aTransferPackages[5].iAddressedTarget := 12;
		aTransferPackages[5].iIndex := 21;
		
	//iVolumeAt2
		aTransferPackages[6].iChannel := iParameterSet;
		aTransferPackages[6].iAddressedTarget := 12;
		aTransferPackages[6].iIndex := 40;
		
	//iVolumeAt4 
		aTransferPackages[7].iChannel := iParameterSet;
		aTransferPackages[7].iAddressedTarget := 12;
		aTransferPackages[7].iIndex := 41;
		
	//iInstallationPositionDrive
		aTransferPackages[8].iChannel := iParameterSet;
		aTransferPackages[8].iAddressedTarget := 12;
		aTransferPackages[8].iIndex := 60;
		
	//iLoadRetracting
		aTransferPackages[9].iChannel := iParameterSet;
		aTransferPackages[9].iAddressedTarget := 12;
		aTransferPackages[9].iIndex := 100;
		
	//iLoadAdvancing
		aTransferPackages[10].iChannel := iParameterSet;
		aTransferPackages[10].iAddressedTarget := 12;
		aTransferPackages[10].iIndex := 101;
		
	//iMomentOfInertiaRetracting
		aTransferPackages[11].iChannel := iParameterSet;
		aTransferPackages[11].iAddressedTarget := 12;
		aTransferPackages[11].iIndex := 102;
		
	//iMomentOfInertiaAdvancing
		aTransferPackages[12].iChannel := iParameterSet;
		aTransferPackages[12].iAddressedTarget := 12;
		aTransferPackages[12].iIndex := 103;
		
	//iMaxLeakageForStatusGood
		aTransferPackages[13].iChannel := iParameterSet;
		aTransferPackages[13].iAddressedTarget := 12;
		aTransferPackages[13].iIndex := 200;
		
	//iMaxLeakageForStatusWarning
		aTransferPackages[14].iChannel := iParameterSet;
		aTransferPackages[14].iAddressedTarget := 12;
		aTransferPackages[14].iIndex := 201;
		
	//iMaxLeakageForStatusCritical
		aTransferPackages[15].iChannel := iParameterSet;
		aTransferPackages[15].iAddressedTarget := 12;
		aTransferPackages[15].iIndex := 202;
		
	// define end of parameter list to be uploaded by setting all variables to 0 (end criterion for FB_Upload_Multiple_Parameters)
		aTransferPackages[16].iChannel := 0;
		aTransferPackages[16].iAddressedTarget := 0;
		aTransferPackages[16].iIndex := 0;
//-----------------------------------------------------------------------------------------------------------

// Read the current status of the the motion terminal
	fbreadbitsfromword(wData:= awBusDataFromVTEM[0], iStartBit:=0, iEndBit:= 5, iValue=> iCurrentValveMode, xError=> );				// read current valve mode
//-----------------------------------------------------------------------------------------------------------

// Transition: Aborting condition when xAbort is TRUE in all States except "IDLE" , "ABORTING" and "RESETTING"
	IF xAbort = TRUE AND NOT(iState = 10 AND xExecute = FALSE) AND iState <> 80 AND iState <> 100 THEN
		xStateChange := TRUE;	// Leaving current state
		iState := 80;	// Choosing next state, here: ABORTING
	END_IF
//-----------------------------------------------------------------------------------------------------------

// local state machine
	CASE iState OF
		10:	// IDLE
			// code that is executed only in the first cycle of this state
				IF xStateChange = TRUE THEN
					xStateChange := FALSE;
					iResponse := eTransferResponse.ready_for_new_transfer;
					xDone := FALSE;
					xError := FALSE;
					xBusy := FALSE;
					xAborted := FALSE;
				END_IF
			//-----------------------------------------------------------------------------------------------------------
			
			// code that is repeated every cycle in this state
				iCommandNumber := 0;
			//-----------------------------------------------------------------------------------------------------------
			
			// Transition
			IF xExecute = TRUE THEN
				xStateChange := TRUE;
				iState := 20;
			END_IF
			//-----------------------------------------------------------------------------------------------------------
		
		20:	// RESETTING VALVE MODE TO 61
			// code that is executed only in the first cycle of this state
				IF xStateChange = TRUE THEN
					xStateChange := FALSE;
					iResponse := eTransferResponse.preparing_transfer;
					xDone := FALSE;
					xError := FALSE;
					xBusy := TRUE;
					xAborted := FALSE;
				END_IF
			//-----------------------------------------------------------------------------------------------------------
			
			// code that is repeated every cycle in this state	
				IF iCurrentValveMode = 63 THEN
					iCommandNumber := 5;	// exit transfer mode
				ELSIF iCurrentValveMode <> 61 AND iCurrentValveMode <> 63 THEN
					iCommandNumber := 6;	// stop running motion apps
				END_IF 
			//-----------------------------------------------------------------------------------------------------------
			
			// Transition
				IF iCurrentValveMode = 61 THEN
					xStateChange := TRUE;	// Leave this state
					iState := 30;
					iCommandNumber := 30;			
				END_IF
			//-----------------------------------------------------------------------------------------------------------
		
		30:	// READING PARAMETER VALUES
			// code that is executed only in the first cycle of this state
				IF xStateChange = TRUE THEN
					xStateChange := FALSE;
					iResponse := eTransferResponse.transferring;
					xDone := FALSE;
					xError := FALSE;
					xBusy := TRUE;
					xAborted := FALSE;
				END_IF
			//-----------------------------------------------------------------------------------------------------------
			
			// code that is repeated every cycle in this state
				iCommandNumber := 30;		// read parameter values
			//-----------------------------------------------------------------------------------------------------------
			
			// Transition
				IF fbuploadMultipleParameters.xExecute = TRUE AND fbuploadMultipleParameters.xUploadDone = TRUE AND fbuploadMultipleParameters.xUploadError = FALSE THEN	// Upload Done
					xStateChange := TRUE;
					iState := 40;	// Write parameter values to outputs
				ELSIF fbuploadMultipleParameters.xExecute = TRUE AND fbuploadMultipleParameters.xUploadDone = FALSE AND fbuploadMultipleParameters.xUploadError = TRUE THEN	// Error during update
					xStateChange := TRUE;
					iState := 70;	// ERROR
					iResponse := fbuploadMultipleParameters.iResponse;
				END_IF
			//-----------------------------------------------------------------------------------------------------------
		
		40:	// WRITE PARAMETER VALUES TO OUTPUTS
			// code that is executed only in the first cycle of this state
				IF xStateChange = TRUE THEN
					xStateChange := FALSE;
					iResponse := eTransferResponse.transferring;
					xDone := FALSE;
					xError := FALSE;
					xBusy := TRUE;
					xAborted := FALSE;
				END_IF
			//-----------------------------------------------------------------------------------------------------------
			
			// code that is repeated every cycle in this state
				iTubingLengthAt2				:= aTransferPackages[0].iTransferValue;
				iTubingLengthAt4				:= aTransferPackages[1].iTransferValue;
				iTubingInnerDiameterAt2			:= aTransferPackages[2].iTransferValue;
				iTubingInnerDiameterAt4			:= aTransferPackages[3].iTransferValue;
				iDriveType						:= aTransferPackages[4].iTransferValue;
				iDriveStroke					:= aTransferPackages[5].iTransferValue;
				iVolumeAt2						:= aTransferPackages[6].iTransferValue;
				iVolumeAt4						:= aTransferPackages[7].iTransferValue;
				iInstallationPositionDrive		:= aTransferPackages[8].iTransferValue;
				iLoadRetracting					:= aTransferPackages[9].iTransferValue;
				iLoadAdvancing					:= aTransferPackages[10].iTransferValue;
				iMomentOfInertiaRetracting		:= aTransferPackages[11].iTransferValue;
				iMomentOfInertiaAdvancing		:= aTransferPackages[12].iTransferValue;
				iMaxLeakageForStatusGood		:= aTransferPackages[13].iTransferValue;
				iMaxLeakageForStatusWarning		:= aTransferPackages[14].iTransferValue;
				iMaxLeakageForStatusCritical	:= aTransferPackages[15].iTransferValue;
			//-----------------------------------------------------------------------------------------------------------
			
			// Transition
				xStateChange := TRUE;
				iState := 50;
				iCommandNumber := 40;
			//-----------------------------------------------------------------------------------------------------------
		
		50:	// DONE
			// code that is executed only in the first cycle of this state
				IF xStateChange = TRUE THEN
					xStateChange := FALSE;
					iResponse := eTransferResponse.transfer_successful;
					xDone := TRUE;
					xError := FALSE;
					xBusy := FALSE;
					xAborted := FALSE;
				END_IF
			//-----------------------------------------------------------------------------------------------------------
			
			// code that is repeated every cycle in this state	
				IF fbuploadMultipleParameters.xExecute = FALSE  AND fbuploadMultipleParameters.xUploadDone = FALSE AND fbuploadMultipleParameters.xUploadError = FALSE AND iCurrentValveMode = 63 THEN		//FB_UploadMultipleParameters was reset
					iCommandNumber := 5;	// exit transfer mode
				END_IF
			//-----------------------------------------------------------------------------------------------------------
			
			// Transition
				IF fbuploadMultipleParameters.xExecute = FALSE  AND fbuploadMultipleParameters.xUploadDone = FALSE AND fbuploadMultipleParameters.xUploadError = FALSE AND xExecute = FALSE THEN
					xStateChange := TRUE;
					iState := 100;
				END_IF
			//-----------------------------------------------------------------------------------------------------------
			
		70:	// ERROR
			// code that is executed only in the first cycle of this state
				IF xStateChange = TRUE THEN
					xStateChange := FALSE;
					//iResponse := eTransferResponse.communication_failed;	// set within the transition of the last state
					xDone := FALSE;
					xError := TRUE;
					xBusy := FALSE;
					xAborted := FALSE;
				END_IF
			//-----------------------------------------------------------------------------------------------------------
			
			// code that is repeated every cycle in this state	
			//-----------------------------------------------------------------------------------------------------------
			
			// Transition
				IF xExecute = FALSE AND xAbort = FALSE THEN
					xStateChange := TRUE;
					iState := 100;
				END_IF
			//-----------------------------------------------------------------------------------------------------------
			
		80:	// ABORTING
			// code that is executed only in the first cycle of this state
				IF xStateChange = TRUE THEN
					xStateChange := FALSE;
					iResponse := eTransferResponse.aborting;
					xBusy := FALSE;
					xDone := FALSE;
					xError := FALSE;
					xAborted := TRUE;
				END_IF
			//-----------------------------------------------------------------------------------------------------------
			
			// code that is repeated every cycle in this state
				IF iCurrentValveMode = 63 THEN
					iCommandNumber := 5;	// exit transfer mode
				ELSIF iCurrentValveMode <> 61 AND iCurrentValveMode <> 63 THEN
					iCommandNumber := 6;	// stop running motion apps
				ELSE
					iCommandNumber := 0; 
				END_IF
			//-----------------------------------------------------------------------------------------------------------
			
			// Transition
				IF xAbort = FALSE AND xExecute = FALSE AND iCurrentValveMode = 61 THEN
					xStateChange := TRUE;
					iState := 100;
				END_IF
			//-----------------------------------------------------------------------------------------------------------

		100:	// RESETTING FUNCTION BLOCK AND VALVE
			// code that is executed only in the first cycle of this state
				IF xStateChange = TRUE THEN
					xStateChange := FALSE;
					iResponse := eTransferResponse.resetting;
					xDone := FALSE;
					xError := FALSE;
					xBusy := FALSE;
					xAborted := FALSE;
				END_IF
			//-----------------------------------------------------------------------------------------------------------
			
			// code that is repeated every cycle in this state	
				IF iCurrentValveMode = 63 THEN
					iCommandNumber := 5;	// exit transfer mode
				ELSIF iCurrentValveMode <> 61 AND iCurrentValveMode <> 63 THEN
					iCommandNumber := 6;	// stop running motion apps
				END_IF
				
				// reset funktion block fbreadmultipleparameters
				// not done via command number because this is used to reset valve
					fbuploadMultipleParameters(
						awBusDataFromVTEM:= awBusDataFromVTEM, 
						awBusDataToVTEM:= awBusDataToVTEM, 
						xExecute:= FALSE, 
						iResponse=> , 
						iCurrentValue=> , 
						xUploadDone=> , 
						xUploadError=> , 
						aTransferPackages:= aTransferPackages);
				
				// reset parameter outputs
					iParameterSet					:= 1;

					iTubingLengthAt2				:= 0;
					iTubingLengthAt4				:= 0;
					iTubingInnerDiameterAt2			:= 0;
					iTubingInnerDiameterAt4			:= 0;
					iDriveType						:= 0;
					iDriveStroke					:= 0;
					iVolumeAt2						:= 0;
					iVolumeAt4						:= 0;
					iInstallationPositionDrive		:= 0;
					iLoadRetracting					:= 0;
					iLoadAdvancing					:= 0;
					iMomentOfInertiaRetracting		:= 0;
					iMomentOfInertiaAdvancing		:= 0;
					iMaxLeakageForStatusGood		:= 0;
					iMaxLeakageForStatusWarning		:= 0;
					iMaxLeakageForStatusCritical	:= 0;
				
				// reset parameter array
					FOR iCounterResetArray := 0 TO 100 BY 1 DO
						aTransferPackages[iCounterResetArray].iChannel := 0;
						aTransferPackages[iCounterResetArray].iAddressedTarget := 0;
						aTransferPackages[iCounterResetArray].iIndex := 0;
						aTransferPackages[iCounterResetArray].iTransferValue := 0;
					END_FOR
					
					iCounterResetArray := 0;
					xFirstCycle := TRUE;
			//-----------------------------------------------------------------------------------------------------------
			
			// Transition
				IF iCurrentValveMode = 61 THEN
					iCommandNumber := 6; // Last command to send before the FB is in IDLE
					xStateChange := TRUE;
					iState := 10;
				END_IF
			//-----------------------------------------------------------------------------------------------------------
			
	END_CASE
//-----------------------------------------------------------------------------------------------------------

// Command section
	CASE iCommandNumber OF
		0:	// IDLE
			;
		
		5:	// EXIT TRANSFER MODE
			fbwritevaluetoword(iValue:=63, iStartBit:=0, iEndBit:=5, wDataWord:=awBusDataToVTEM[0], xError=> );							// Valve Mode = 63
			fbwritevaluetoword(iValue:=0, iStartBit:=6, iEndBit:=7, wDataWord:=awBusDataToVTEM[0], xError=> );							// 0 (unused)
			fbwritevaluetoword(iValue:=0, iStartBit:=8, iEndBit:=12, wDataWord:=awBusDataToVTEM[0], xError=> );							// Channel = 0 (ignored)
			fbwritevaluetoword(iValue:=3, iStartBit:=13, iEndBit:=15, wDataWord:=awBusDataToVTEM[0], xError=> );						// Transfer Control = 3 (Exit transfer mode)
			fbwritevaluetoword(iValue:=0, iStartBit:=0, iEndBit:=7, wDataWord:=awBusDataToVTEM[1], xError=> );							// Addressed Target = 0 (ignored)
			fbwritevaluetoword(iValue:=0, iStartBit:=8, iEndBit:=15, wDataWord:=awBusDataToVTEM[1], xError=> );							// Index = 0 (ignored)
			fbwritevaluetoword(iValue:=0, iStartBit:=0, iEndBit:=15, wDataWord:=awBusDataToVTEM[2], xError=> );							// Value = 0 (ignored)
			
		6:	// STOP RUNNING MOTION APP
			fbwritevaluetoword(iValue:=61, iStartBit:=0, iEndBit:=5, wDataWord:=awBusDataToVTEM[0], xError=> );							// Valve Mode = 61 (stop)
			fbwritevaluetoword(iValue:=0, iStartBit:=6, iEndBit:=7, wDataWord:=awBusDataToVTEM[0], xError=> );							// App Control = 0 (unused)
			fbwritevaluetoword(iValue:=0, iStartBit:=8, iEndBit:=15, wDataWord:=awBusDataToVTEM[0], xError=> );							// App Option = 0 (unused)
			fbwritevaluetoword(iValue:=0, iStartBit:=0, iEndBit:=15, wDataWord:=awBusDataToVTEM[1], xError=> );							// Setpoint Value 1 = 0 (unused)
			fbwritevaluetoword(iValue:=0, iStartBit:=0, iEndBit:=15, wDataWord:=awBusDataToVTEM[2], xError=> );							// Setpoint Value 2 = 0 (unused)
		
		30:	// RUN FB_UPLOADMULTIPLEPARAMETERS
			fbuploadMultipleParameters(
				awBusDataFromVTEM:= awBusDataFromVTEM, 
				awBusDataToVTEM:= awBusDataToVTEM, 
				xExecute:= TRUE, 
				iResponse=> , 
				iCurrentValue=> , 
				xUploadDone=> , 
				xUploadError=> , 
				aTransferPackages:= aTransferPackages);

		40:	// RESET FB_UPLOADMULTIPLEPARAMETERS
			fbuploadMultipleParameters(
				awBusDataFromVTEM:= awBusDataFromVTEM, 
				awBusDataToVTEM:= awBusDataToVTEM, 
				xExecute:= FALSE, 
				iResponse=> , 
				iCurrentValue=> , 
				xUploadDone=> , 
				xUploadError=> , 
				aTransferPackages:= aTransferPackages);
	END_CASE
//-----------------------------------------------------------------------------------------------------------

END_FUNCTION_BLOCK

// Transfermode/specific_MA_config/FB_Read_config_MA_33
/// This function block can be used to upload the configuration of Motion App 33 ("Positioning").
/// The specific parameters of this Motion App are the outputs of this FB
/// The function block uses the transfer mode to read this configuration from the Motion Terminal
/// and indicates the state of the upload process at the output iResponse.

FUNCTION_BLOCK FB_Read_config_MA_33
VAR_INPUT
	awBusDataFromVTEM 				: ARRAY [0..2] OF WORD;		// array of 3 words of process data received from the Motion Terminal
END_VAR
	
VAR_IN_OUT
	awBusDataToVTEM 				: ARRAY [0..2] OF WORD; 	// array of 3 words of process data sent to the Motion Terminal
END_VAR

VAR_INPUT
	xExecute 						: BOOL; 					// rising edge starts the reading process, falling edge resets the function block after reading is done
	xAbort							: BOOL;						// rising edge aborts the reading process
	iParameterSet					: INT := 1; 				// the parameter set to be read from, 1 by default
END_VAR                     		

VAR_OUTPUT                  		
	// system parameters
		iTubingLengthAt2 								: INT; 			// length of the tubing connected to outlet port 2 of the valve [1 digit = 1 mm]
	 	iTubingLengthAt4 								: INT;			// length of the tubing connected to outlet port 4 of the valve [1 digit = 1 mm]
	 	iTubingInnerDiameterAt2							: INT;  		// inner diameter of the tubing connected to outlet port 2 of the valve [1 digit = 0.01 mm]
	 	iTubingInnerDiameterAt4							: INT;			// inner diameter of the tubing connected to outlet port 4 of the valve [1 digit = 0.01 mm]
	 	iDriveType 										: INT;			// type of the drive/cylinder/... that is to be operated by the valve ->  see list of drive types at support portal (www.festo.com/sp/)
	 	iDriveStroke 									: INT; 			// stroke of the drive/cylinder/... that is to be operated by the valve [1 digit = 1 mm for linear drives, 1 digit = 1° for rotary drives]
		iInstallationPositionDrive 						: INT;  	 	// inclination of the cylinder with reference to a horizontal installation position [1 digit = 0.01°, positive values = advancing upwards]
		iOffsetAxisZeroPoint							: INT;			// offset of the mechanical stop "retracted" to the retracted end of the nominal stroke [1 digit = 1 mm]
		iInPortFullStrokeMeas							: INT;			// sensor port for positioning measurement over the entire working stroke; value is number of the slot (beginning from 0 and including valve slots) * 10 + number of the port, -1 for usage of partial stroke measurement   
		iInPortPartStrokeMeasRet						: INT;			// sensor port for position measurement over the part of the working stroke at the retracted end; value is number of the slot (beginning from 0 and including valve slots) * 10 + number of the port, -1 if no sensor is connected
		iInPortPartStrokeMeasAdv						: INT;			// sensor port for position measurement over the part of the working stroke at the advanced end; value is number of the slot (beginning from 0 and including valve slots) * 10 + number of the port, -1 if no sensor is connected
	
	// application parameters                               	
		iLoad			 								: INT;			// mass that is to be moved by the drive (retracting and advancing) [1 digit = 0.01 kg]
		iDampingTimeForTargetPositionReached			: INT;			// condition for feedback "Target position reached": actual position remains within the tolerance range around the target position for the specified time [1 digit = 0.01 s]
		iDurationOfThresholdExceedanceForError			: INT;			// condition for following error: Threshold value is exceeded for longer than the configured duration [1 digit = 0.001 s]
		iToleranceForTargetPositionReached				: INT;			// condition for feedback "Target Position Reached": permissible deviation of the actual position from the target position [1 digit = 0.1 mm]
		iMaxVelocityGeneral			 					: INT;			// maximum permissible velocity, independent of the direction of movement (general limitation; further limiting by setpoint value) [1 digit = 0.01 m/s]
		iMaxAcceleration								: INT;			// maximum permissible acceleration in direction of movement [1 digit = 0.1 m/s²]
		iMaxDeceleration								: INT;			// maximum permissible acceleration against the direction of movement [1 digit = 0.1 m/s²]
		iMaxJerk										: INT;			// maximum permissible jerk in direction of movement [1 digit = 0.1 m/s³]
		iOffsetProjectZeroPoint							: INT;			// offset to the reference point for target and actual positions to the axis zero point [1 digit = 1 mm]
		iOffsetSoftLimitNegEndRet						: INT;			// offset to lower "stop" of the desired working stroke to the axis zero point [1 digit = 1 mm]
		iOffsetSoftLimitPosEndAdv						: INT;			// offset to upper "stop" of the desired working stroke to the axis zero point  [1 digit = 1 mm]

		iDistTargPosWithConstVeloRet					: INT;			// Contact case: Distance to target position in retracting direction, on which the configured final velocity is to be applied
		iFinalVeloContactCaseRet						: INT;			// Contact case: Final velocity at contact in retracting direction
		iDistTargPosWithConstVeloAdv					: INT;			// Contact case: Distance to target position in advancing direction, on which the configured final velocity is to be applied
		iFinalVeloContactCaseAdv						: INT;			// Contact case: Final velocity at contact in advancing direction

		iMeanPressureLevel								: INT;			// mean pressure level [1 digit = 0.1 bar rel.]
		iThreshPosFollowError							: INT; 			// condition for following error: Actual position deviates from the planned trajectory by more than the threshold value for at least the configured duration [1 digit = 1 mm]  
		iTreshVeloFollowError							: INT; 			// condition for following error: Actual velocity deviates from the planned trajectory by more than the threshold value for at least the configured duration [1 digit = 0.001 m/s]
		iSoftStartFunction								: INT;			// Pre-pressurisation of cylinder chambers; 0 = disabled, 1 = enabled
		iEndPositionMonitoring							: INT;			// 0 = active for both end positions, 1 = active for retracted end position, 2 = active for advanced end position, 3 = inactive 
		xOptionPressureBuildUpIntoMechEndPos			: BOOL;			// 0 = Setpoint values are only accepted within the actual effective stroke, 1 = Allow setpoint values outside the actual effective stroke in order to build up pressure into the mechanical end position

	// tuning parameters
		iOptControllerGainRelative						: INT;			// Optional tuning parameter for controller gain (relative adjustment of the internally used value) [1 digit = 1%]
		iOptDampingOfSystemAbsolute						: INT;			// Optional tuning parameter for damping of the controlled system (absolute adjustment of the internally used value [1 digit = 0.01]
		iOptPliabilityRelative							: INT;			// Optional tuning parameter for pliability (relative adjustment of the internally used value) [1 digit = 1%]
		iOptReductionOfPilotControlRelative				: INT;			// Optional tuning parameter for reduction of pilot control (relative adjustment of the internally used value) [1 digit = 1%]
		iOptCoulombFritionInAccountRelative				: INT;			// Optional tuning parameter for coulomb friction taken into account(relative adjustment of the internally used value) [1 digit = 1%]
		
	// function block response
		iResponse 					: eTransferResponse; 		// returns the status of the upload process
		xBusy						: BOOL;						// TRUE as long as the upload process is running
		xDone 						: BOOL; 					// indicates whether the upload was successfull
		xError 						: BOOL; 					// indicates whether an error occurred during the transfer
		xAborted					: BOOL;						// TRUE if the function block was canceled by xAbort	
END_VAR

VAR
	iState							: INT := 10;
	xStateChange					: BOOL;
	iCommandNumber					: INT;
	xFirstCycle						: BOOL := TRUE;				// indicator for the first cycle of the function block
	iParameterSetFC					: INT;						// value on input iParameterSet during first cycle
	
	aTransferPackages				: ARRAY [0..100] OF stTransferPackage;
	fbreadbitsfromword				: FB_Read_Bits_From_Word;
	fbuploadMultipleParameters 		: FB_Upload_Multiple_Parameters;
	fbWriteValueToWord 				: FB_Write_Value_To_Word;

	iCounterResetArray				: INT;

	iCurrentValveMode				: INT;						//
END_VAR

(*****************************************************************************************************

Festo SE & Co. KG, Esslingen
Copyright (c) 2021. All rights reserved.

Product:            Motion Terminal VTEM
Description:        Function Block to upload the parameters for Motion App 33 from the Motion Terminal

Object version:     2.00
Last change:        2021-07
======================================================================================================
                                       H I S T O R Y
======================================================================================================
Version:            2.00
Date:               2021-07
Change/Activity:    - created (#3872357)
Release:            3.5.7.237 (CODESYS 3.5.7.2, Lib version 3.7)
Author:             JEBU
======================================================================================================

*****************************************************************************************************)

// pre-check of the value for the parameter set
	IF xExecute = TRUE AND (iParameterSet < 1 OR iParameterSet > 5) THEN		// invalid input for the parameter set
		xDone := FALSE; 
		xError := TRUE; 
		iResponse := eTransferResponse.invalid_ParameterSet;
		xStateChange := TRUE;
		iState := 70;	// ERROR
	END_IF
//-----------------------------------------------------------------------------------------------------------

// check if iParameterSet was changed
	IF xExecute = TRUE AND xFirstCycle = TRUE THEN
		xFirstCycle := FALSE;
		iParameterSetFC := iParameterSet;
	END_IF
	
	IF xExecute = TRUE AND iParameterSet <> iParameterSetFC THEN
		xStateChange := TRUE;
		iState := 70;
		iResponse := eTransferResponse.FB_needs_rising_edge_xExecute;
	END_IF
//-----------------------------------------------------------------------------------------------------------

// WRITE PARAMETER INDICES INTO ARRAY
	//iTubingLengthAt2
		aTransferPackages[0].iChannel := iParameterSet;
		aTransferPackages[0].iAddressedTarget := 33;
		aTransferPackages[0].iIndex := 12;
		
	//iTubingLengthAt4
		aTransferPackages[1].iChannel := iParameterSet;
		aTransferPackages[1].iAddressedTarget := 33;
		aTransferPackages[1].iIndex := 13;
		
	//iTubingInnerDiameterAt2
		aTransferPackages[2].iChannel := iParameterSet;
		aTransferPackages[2].iAddressedTarget := 33;
		aTransferPackages[2].iIndex := 14;
		
	//iTubingInnerDiameterAt4
		aTransferPackages[3].iChannel := iParameterSet;
		aTransferPackages[3].iAddressedTarget := 33;
		aTransferPackages[3].iIndex := 15;
		
	//iDriveType
		aTransferPackages[4].iChannel := iParameterSet;
		aTransferPackages[4].iAddressedTarget := 33;
		aTransferPackages[4].iIndex := 20;
		
	//iDriveStroke
		aTransferPackages[5].iChannel := iParameterSet;
		aTransferPackages[5].iAddressedTarget := 33;
		aTransferPackages[5].iIndex := 21;
		
	//iInstallationPositionDrive
		aTransferPackages[6].iChannel := iParameterSet;
		aTransferPackages[6].iAddressedTarget := 33;
		aTransferPackages[6].iIndex := 60;
		
	//iOffsetAxisZeroPoint
		aTransferPackages[7].iChannel := iParameterSet;
		aTransferPackages[7].iAddressedTarget := 33;
		aTransferPackages[7].iIndex := 61;
		
	//iInPortFullStrokeMeas
		aTransferPackages[8].iChannel := iParameterSet;
		aTransferPackages[8].iAddressedTarget := 33;
		aTransferPackages[8].iIndex := 80;
		
	//iInPortPartStrokeMeasRet
		aTransferPackages[9].iChannel := iParameterSet;
		aTransferPackages[9].iAddressedTarget := 33;
		aTransferPackages[9].iIndex := 75;
		
	//iInPortPartStrokeMeasAdv
		aTransferPackages[10].iChannel := iParameterSet;
		aTransferPackages[10].iAddressedTarget := 33;
		aTransferPackages[10].iIndex := 76;
		
	//iLoad
		aTransferPackages[11].iChannel := iParameterSet;
		aTransferPackages[11].iAddressedTarget := 33;
		aTransferPackages[11].iIndex := 100;
		
	//iDampingTimeForTargetPositionReached
		aTransferPackages[12].iChannel := iParameterSet;
		aTransferPackages[12].iAddressedTarget := 33;
		aTransferPackages[12].iIndex := 124;
		
	//iDurationOfThresholdExceedanceForError
		aTransferPackages[13].iChannel := iParameterSet;
		aTransferPackages[13].iAddressedTarget := 33;
		aTransferPackages[13].iIndex := 126;
		
	//iToleranceForTargetPositionReached	
		aTransferPackages[14].iChannel := iParameterSet;
		aTransferPackages[14].iAddressedTarget := 33;
		aTransferPackages[14].iIndex := 141;
		
	// iMaxVelocityGeneral
		aTransferPackages[15].iChannel := iParameterSet;
		aTransferPackages[15].iAddressedTarget := 33;
		aTransferPackages[15].iIndex := 142;
		
	//iMaxAcceleration
		aTransferPackages[16].iChannel := iParameterSet;
		aTransferPackages[16].iAddressedTarget := 33;
		aTransferPackages[16].iIndex := 144;
		
	//iMaxDecelaration
		aTransferPackages[17].iChannel := iParameterSet;
		aTransferPackages[17].iAddressedTarget := 33;
		aTransferPackages[17].iIndex := 146;
		
	//iMaxJerk
		aTransferPackages[18].iChannel := iParameterSet;
		aTransferPackages[18].iAddressedTarget := 33;
		aTransferPackages[18].iIndex := 148;
		
	//iOffsetProjectZeroPoint
		aTransferPackages[19].iChannel := iParameterSet;
		aTransferPackages[19].iAddressedTarget := 33;
		aTransferPackages[19].iIndex := 150;
		
	//iOffsetSoftLimitNegEndRet
		aTransferPackages[20].iChannel := iParameterSet;
		aTransferPackages[20].iAddressedTarget := 33;
		aTransferPackages[20].iIndex := 151;
		
	//iOffsetSoftLimitPosEndAdv
		aTransferPackages[21].iChannel := iParameterSet;
		aTransferPackages[21].iAddressedTarget := 33;
		aTransferPackages[21].iIndex := 152;
		
	//iDistTargPosWithConstVeloRet
		aTransferPackages[22].iChannel := iParameterSet;
		aTransferPackages[22].iAddressedTarget := 33;
		aTransferPackages[22].iIndex := 153;
		
	//iFinalVeloContactCaseRet
		aTransferPackages[23].iChannel := iParameterSet;
		aTransferPackages[23].iAddressedTarget := 33;
		aTransferPackages[23].iIndex := 155;
		
	//iDistTargPosWithConstVeloAdv
		aTransferPackages[24].iChannel := iParameterSet;
		aTransferPackages[24].iAddressedTarget := 33;
		aTransferPackages[24].iIndex := 154;
		
